HMI tags "2080SP242U01"
   "2080SP242U01.AI1" : Real AT %DB4304.DBD6, 500 ms
   "2080SP242U01.AI2" : Real AT %DB4304.DBD10, 500 ms
   "2080SP242U01.AI3" : Real AT %DB4304.DBD14, 500 ms
   "2080SP242U01.AO1a" : Real AT %DB4304.DBD34, 500 ms
   "2080SP242U01.AO1b" : Real AT %DB4304.DBD38, 500 ms
   "2080SP242U01.AO2a" : Real AT %DB4304.DBD42, 500 ms
   "2080SP242U01.AO2b" : Real AT %DB4304.DBD42, 500 ms
   "2080SP242U01.AO3a" : Real AT %DB4304.DBD50, 500 ms
   "2080SP242U01.AO3b" : Real AT %DB4304.DBD46, 500 ms
   "2080SP242U01.BlockInfo" : Array [0..4] of Int AT %DB4304.DBX74.0, 500 ms
   "2080SP242U01.DefaultText" : TextRef, internal   // Заголовок POPUP окна. При експорте из ECS через скрипт заполняется автоматически, если теги копируются в ручную то требуется в ручную задатать свойство Start Value
   "2080SP242U01.DI.ACK" : Bool AT %DB4304.DBX5.3, 500 ms
   "2080SP242U01.DI.ASTR" : Bool AT %DB4304.DBX2.1, 500 ms
   "2080SP242U01.DI.BUSF" : Bool AT %DB4304.DBX4.5, 500 ms
   "2080SP242U01.DI.DIR" : Bool AT %DB4304.DBX2.2, 500 ms
   "2080SP242U01.DI.DOPR" : Bool AT %DB4304.DBX4.6, 500 ms
   "2080SP242U01.DI.DRDY" : Bool AT %DB4304.DBX3.6, 500 ms
   "2080SP242U01.DI.DTEST" : Bool AT %DB4304.DBX4.7, 500 ms
   "2080SP242U01.DI.EARTH" : Bool AT %DB4304.DBX4.1, 500 ms
   "2080SP242U01.DI.ES" : Bool AT %DB4304.DBX5.2, 500 ms
   "2080SP242U01.DI.GFA" : Bool AT %DB4304.DBX4.3, 500 ms
   "2080SP242U01.DI.GWA" : Bool AT %DB4304.DBX4.4, 500 ms
   "2080SP242U01.DI.LSTP" : Bool AT %DB4304.DBX3.2, 500 ms
   "2080SP242U01.DI.LSTR1" : Bool AT %DB4304.DBX3.0, 500 ms
   "2080SP242U01.DI.LSTR2" : Bool AT %DB4304.DBX3.1, 500 ms
   "2080SP242U01.DI.MCC" : Bool AT %DB4304.DBX2.3, 500 ms
   "2080SP242U01.DI.MD" : Bool AT %DB4304.DBX3.7, 500 ms
   "2080SP242U01.DI.OVL" : Bool AT %DB4304.DBX2.5, 500 ms
   "2080SP242U01.DI.RDY" : Bool AT %DB4304.DBX2.4, 500 ms
   "2080SP242U01.DI.REM" : Bool AT %DB4304.DBX3.3, 500 ms
   "2080SP242U01.DI.RET1" : Bool AT %DB4304.DBX2.6, 500 ms
   "2080SP242U01.DI.RET2" : Bool AT %DB4304.DBX2.7, 500 ms
   "2080SP242U01.DI.SEL" : Bool AT %DB4304.DBX2.0, 500 ms
   "2080SP242U01.DI.SFS" : Bool AT %DB4304.DBX5.0, 500 ms
   "2080SP242U01.DI.SLS" : Bool AT %DB4304.DBX5.1, 500 ms
   "2080SP242U01.DI.SSW" : Bool AT %DB4304.DBX3.4, 500 ms
   "2080SP242U01.DI.STALL" : Bool AT %DB4304.DBX4.0, 500 ms
   "2080SP242U01.DI.TFA" : Bool AT %DB4304.DBX3.5, 500 ms
   "2080SP242U01.DI.UBAL" : Bool AT %DB4304.DBX4.2, 500 ms
   "2080SP242U01.DQ.ASTW" : Bool AT %DB4304.DBX32.0, 500 ms
   "2080SP242U01.DQ.AUT" : Bool AT %DB4304.DBX31.4, 500 ms
   "2080SP242U01.DQ.CON1" : Bool AT %DB4304.DBX30.0, 500 ms
   "2080SP242U01.DQ.CON2" : Bool AT %DB4304.DBX30.1, 500 ms
   "2080SP242U01.DQ.LAMP1" : Bool AT %DB4304.DBX30.2, 500 ms
   "2080SP242U01.DQ.LAMP2" : Bool AT %DB4304.DBX30.3, 500 ms
   "2080SP242U01.DQ.LOC" : Bool AT %DB4304.DBX31.2, 500 ms
   "2080SP242U01.DQ.MAN" : Bool AT %DB4304.DBX31.3, 500 ms
   "2080SP242U01.DQ.OK" : Bool AT %DB4304.DBX31.1, 500 ms
   "2080SP242U01.DQ.RD1" : Bool AT %DB4304.DBX30.5, 500 ms
   "2080SP242U01.DQ.RD2" : Bool AT %DB4304.DBX30.6, 500 ms
   "2080SP242U01.DQ.RES" : Bool AT %DB4304.DBX31.6, 500 ms
   "2080SP242U01.DQ.RUN1" : Bool AT %DB4304.DBX30.7, 500 ms
   "2080SP242U01.DQ.RUN2" : Bool AT %DB4304.DBX31.0, 500 ms
   "2080SP242U01.DQ.SACK" : Bool AT %DB4304.DBX30.4, 500 ms
   "2080SP242U01.DQ.SS" : Bool AT %DB4304.DBX31.5, 500 ms
   "2080SP242U01.DQ.TESTP" : Bool AT %DB4304.DBX31.7, 500 ms
   "2080SP242U01.FP_CMD" : Int AT %DB4304.DBW84, 500 ms
   "2080SP242U01.FP_CMD.AckAlarm" : Bool AT %DB4304.DBX84.7, 500 ms
   "2080SP242U01.FP_CMD.Auto" : Bool AT %DB4304.DBX85.0, 500 ms
   "2080SP242U01.FP_CMD.Local" : Bool AT %DB4304.DBX85.2, 500 ms
   "2080SP242U01.FP_CMD.Manual" : Bool AT %DB4304.DBX85.1, 500 ms
   "2080SP242U01.FP_CMD.QuickStop" : Bool AT %DB4304.DBX84.0, 500 ms
   "2080SP242U01.FP_CMD.Reset" : Bool AT %DB4304.DBX85.6, 500 ms
   "2080SP242U01.FP_CMD.Start1" : Bool AT %DB4304.DBX85.3, 500 ms
   "2080SP242U01.FP_CMD.Start2" : Bool AT %DB4304.DBX85.4, 500 ms
   "2080SP242U01.FP_CMD.Stop" : Bool AT %DB4304.DBX85.5, 500 ms
   "2080SP242U01.FP_CMD.Test" : Bool AT %DB4304.DBX85.7, 500 ms
   "2080SP242U01.FP_DIM.Auto" : Bool AT %DB4304.DBX92.0, 500 ms
   "2080SP242U01.FP_DIM.FP_DIM" : Bool AT %DB4304.DBX92.0, 500 ms
   "2080SP242U01.FP_DIM.Local" : Bool AT %DB4304.DBX92.1, 500 ms
   "2080SP242U01.FP_DIM.Manual" : Bool AT %DB4304.DBX92.2, 500 ms
   "2080SP242U01.FP_DIM.QStop" : Bool AT %DB4304.DBX92.7, 500 ms
   "2080SP242U01.FP_DIM.Reset" : Bool AT %DB4304.DBX93.0, 500 ms
   "2080SP242U01.FP_DIM.Start1" : Bool AT %DB4304.DBX92.3, 500 ms
   "2080SP242U01.FP_DIM.Start2" : Bool AT %DB4304.DBX92.4, 500 ms
   "2080SP242U01.FP_DIM.Stop" : Bool AT %DB4304.DBX92.5, 500 ms
   "2080SP242U01.FP_DIM.TEst" : Bool AT %DB4304.DBX92.6, 500 ms
   "2080SP242U01.FP_DIM1" : Array [0..15] of Bool AT %DB4304.DBX92.0, 500 ms
   "2080SP242U01.FP_EN.Mode_Auto" : Bool AT %DB4304.DBX90.0, 500 ms
   "2080SP242U01.FP_EN.Mode_Loc" : Bool AT %DB4304.DBX90.2, 500 ms
   "2080SP242U01.FP_EN.Mode_Loc_1" : Bool AT %DB4304.DBX90.3, 500 ms
   "2080SP242U01.FP_EN.Mode_Man" : Bool AT %DB4304.DBX90.1, 500 ms
   "2080SP242U01.FP_EN.Mode_SS_Field" : Bool AT %DB4304.DBX90.4, 500 ms
   "2080SP242U01.FP_EN.Mode_SS_FP" : Bool AT %DB4304.DBX90.5, 500 ms
   "2080SP242U01.FP_EN.Mode_Test" : Bool AT %DB4304.DBX90.3, 500 ms
   "2080SP242U01.FP_EN.PB_QStop" : Bool AT %DB4304.DBX90.6, 500 ms
   "2080SP242U01.FP_PARM.AI1_Max" : Real AT %DB4304.DBD158, 500 ms
   "2080SP242U01.FP_PARM.AI1_Min" : Real AT %DB4304.DBD162, 500 ms
   "2080SP242U01.FP_PARM.AI2_Max" : Real AT %DB4304.DBD166, 500 ms
   "2080SP242U01.FP_PARM.AI2_Min" : Real AT %DB4304.DBD170, 500 ms
   "2080SP242U01.FP_PARM.AI3_Max" : Real AT %DB4304.DBD174, 500 ms
   "2080SP242U01.FP_PARM.AI3_Min" : Real AT %DB4304.DBD178, 500 ms
   "2080SP242U01.FP_PARM.AO1a_Max" : Real AT %DB4304.DBD182, 500 ms
   "2080SP242U01.FP_PARM.AO1a_Min" : Real AT %DB4304.DBD186, 500 ms
   "2080SP242U01.FP_PARM.AO1b_Max" : Real AT %DB4304.DBD206, 500 ms
   "2080SP242U01.FP_PARM.AO1b_Min" : Real AT %DB4304.DBD210, 500 ms
   "2080SP242U01.FP_PARM.AO2a_Max" : Real AT %DB4304.DBD190, 500 ms
   "2080SP242U01.FP_PARM.AO2a_Min" : Real AT %DB4304.DBD194, 500 ms
   "2080SP242U01.FP_PARM.AO2b_Max" : Real AT %DB4304.DBD214, 500 ms
   "2080SP242U01.FP_PARM.AO2b_Min" : Real AT %DB4304.DBD218, 500 ms
   "2080SP242U01.FP_PARM.AO3a_Max" : Real AT %DB4304.DBD198, 500 ms
   "2080SP242U01.FP_PARM.AO3a_Min" : Real AT %DB4304.DBD202, 500 ms
   "2080SP242U01.FP_PARM.AO3b_Max" : Real AT %DB4304.DBD222, 500 ms
   "2080SP242U01.FP_PARM.AO3b_Min" : Real AT %DB4304.DBD226, 500 ms
   "2080SP242U01.FP_PARM.ChangeDir_Acc" : Int AT %DB4304.DBW138, 500 ms
   "2080SP242U01.FP_PARM.ChangeDir_Pre" : Int AT %DB4304.DBW136, 500 ms
   "2080SP242U01.FP_PARM.DelayStart_Acc" : Int AT %DB4304.DBW114, 500 ms
   "2080SP242U01.FP_PARM.DelayStart_Pre" : Int AT %DB4304.DBW112, 500 ms
   "2080SP242U01.FP_PARM.DelayStop_Acc" : Int AT %DB4304.DBW118, 500 ms
   "2080SP242U01.FP_PARM.DelayStop_Pre" : Int AT %DB4304.DBW116, 500 ms
   "2080SP242U01.FP_PARM.INTL" : Bool AT %DB4304.DBX230.0, 500 ms
   "2080SP242U01.FP_PARM.INTL_SEQ_STP" : Bool AT %DB4304.DBX230.3, 500 ms
   "2080SP242U01.FP_PARM.INTL_SEQ_STR1" : Bool AT %DB4304.DBX230.1, 500 ms
   "2080SP242U01.FP_PARM.INTL_SEQ_STR2" : Bool AT %DB4304.DBX230.2, 500 ms
   "2080SP242U01.FP_PARM.LeaveFS_Acc" : Int AT %DB4304.DBW142, 500 ms
   "2080SP242U01.FP_PARM.LeaveFS_Pre" : Int AT %DB4304.DBW140, 500 ms
   "2080SP242U01.FP_PARM.MD_Freq_PV" : Int AT %DB4304.DBW154, 500 ms
   "2080SP242U01.FP_PARM.MD_Freq_SP" : Int AT %DB4304.DBW152, 500 ms
   "2080SP242U01.FP_PARM.ReachFS_Acc" : Int AT %DB4304.DBW150, 500 ms
   "2080SP242U01.FP_PARM.ReachFS_Pre" : Int AT %DB4304.DBW148, 500 ms
   "2080SP242U01.FP_PARM.ReachLS_Acc" : Int AT %DB4304.DBW146, 500 ms
   "2080SP242U01.FP_PARM.ReachLS_Pre" : Int AT %DB4304.DBW144, 500 ms
   "2080SP242U01.FP_PARM.ReturnMon_Acc" : Int AT %DB4304.DBW122, 500 ms
   "2080SP242U01.FP_PARM.ReturnMon_Pre" : Int AT %DB4304.DBW120, 500 ms
   "2080SP242U01.FP_PARM.RunDelay1_Acc" : Int AT %DB4304.DBW106, 500 ms
   "2080SP242U01.FP_PARM.RunDelay1_Pre" : Int AT %DB4304.DBW104, 500 ms
   "2080SP242U01.FP_PARM.RunDelay2_Acc" : Int AT %DB4304.DBW110, 500 ms
   "2080SP242U01.FP_PARM.RunDelay2_Pre" : Int AT %DB4304.DBW108, 500 ms
   "2080SP242U01.FP_PARM.SpeedMonOffDelay_Acc" : Int AT %DB4304.DBW130, 500 ms
   "2080SP242U01.FP_PARM.SpeedMonOffDelay_Pre" : Int AT %DB4304.DBW128, 500 ms
   "2080SP242U01.FP_PARM.SpeedMonOnDelay_Acc" : Int AT %DB4304.DBW126, 500 ms
   "2080SP242U01.FP_PARM.SpeedMonOnDelay_Pre" : Int AT %DB4304.DBW124, 500 ms
   "2080SP242U01.FP_PARM.SpeedMonTrigDelay_Acc" : Int AT %DB4304.DBW134, 500 ms
   "2080SP242U01.FP_PARM.SpeedMonTrigDelay_Pre" : Int AT %DB4304.DBW132, 500 ms
   "2080SP242U01.FP_PARM.StartWarn_Acc" : Int AT %DB4304.DBW102, 500 ms
   "2080SP242U01.FP_PARM.StartWarn_Pre" : Int AT %DB4304.DBW100, 500 ms
   "2080SP242U01.FP_PARM.StopReason" : Int AT %DB4304.DBW156, 500 ms
   "2080SP242U01.FP_SEL.INCH_Loc" : Bool AT %DB4304.DBX87.7, 500 ms
   "2080SP242U01.FP_SEL.INCH_Man" : Bool AT %DB4304.DBX87.6, 500 ms
   "2080SP242U01.FP_SEL.MD" : Bool AT %DB4304.DBX86.0, 500 ms
   "2080SP242U01.FP_SEL.MD_Maintain" : Bool AT %DB4304.DBX86.3, 500 ms
   "2080SP242U01.FP_SEL.MD_OnOff" : Bool AT %DB4304.DBX86.2, 500 ms
   "2080SP242U01.FP_SEL.MD_Puls" : Bool AT %DB4304.DBX86.1, 500 ms
   "2080SP242U01.FP_SEL.MotorStarter" : Bool AT %DB4304.DBX87.3, 500 ms
   "2080SP242U01.FP_SEL.OutOfSevice" : Bool AT %DB4304.DBX88.0, 500 ms
   "2080SP242U01.FP_SEL.ParentCollection" : Bool AT %DB4304.DBX87.5, 500 ms
   "2080SP242U01.FP_SEL.ParentSupress" : Bool AT %DB4304.DBX87.4, 500 ms
   "2080SP242U01.FP_SEL.STW_AutoStart" : Bool AT %DB4304.DBX86.4, 500 ms
   "2080SP242U01.FP_SEL.STW_Local" : Bool AT %DB4304.DBX86.5, 500 ms
   "2080SP242U01.FP_SEL.STW_Manual" : Bool AT %DB4304.DBX86.6, 500 ms
   "2080SP242U01.FP_SEL.STW_Single" : Bool AT %DB4304.DBX86.7, 500 ms
   "2080SP242U01.FP_SEL.Type_Bimotor" : Bool AT %DB4304.DBX87.1, 500 ms
   "2080SP242U01.FP_SEL.Type_Indication" : Bool AT %DB4304.DBX87.2, 500 ms
   "2080SP242U01.FP_SEL.Type_Unimotor" : Bool AT %DB4304.DBX87.0, 500 ms
   "2080SP242U01.FP_SEL.WarningDrive" : Bool AT %DB4304.DBX88.1, 500 ms
   "2080SP242U01.FP_SHOW.ACK" : Bool AT %DB4304.DBX97.5, 500 ms
   "2080SP242U01.FP_SHOW.AI1" : Bool AT %DB4304.DBX95.0, 500 ms
   "2080SP242U01.FP_SHOW.AI2" : Bool AT %DB4304.DBX95.1, 500 ms
   "2080SP242U01.FP_SHOW.AI3" : Bool AT %DB4304.DBX95.2, 500 ms
   "2080SP242U01.FP_SHOW.ASTR" : Bool AT %DB4304.DBX99.2, 500 ms
   "2080SP242U01.FP_SHOW.B1" : Byte AT %DB4304.DBB95, 500 ms
   "2080SP242U01.FP_SHOW.B2" : Byte AT %DB4304.DBB96, 500 ms
   "2080SP242U01.FP_SHOW.B3" : Byte AT %DB4304.DBB97, 500 ms
   "2080SP242U01.FP_SHOW.B4" : Byte AT %DB4304.DBB98, 500 ms
   "2080SP242U01.FP_SHOW.BUSF" : Bool AT %DB4304.DBX97.2, 500 ms
   "2080SP242U01.FP_SHOW.ChangeDir" : Bool AT %DB4304.DBX99.0, 500 ms
   "2080SP242U01.FP_SHOW.CON2" : Bool AT %DB4304.DBX98.2, 500 ms
   "2080SP242U01.FP_SHOW.DelayRun2" : Bool AT %DB4304.DBX98.7, 500 ms
   "2080SP242U01.FP_SHOW.DOPR" : Bool AT %DB4304.DBX97.3, 500 ms
   "2080SP242U01.FP_SHOW.DRDY" : Bool AT %DB4304.DBX96.4, 500 ms
   "2080SP242U01.FP_SHOW.DTEST" : Bool AT %DB4304.DBX97.4, 500 ms
   "2080SP242U01.FP_SHOW.EARTH" : Bool AT %DB4304.DBX96.6, 500 ms
   "2080SP242U01.FP_SHOW.ES" : Bool AT %DB4304.DBX96.2, 500 ms
   "2080SP242U01.FP_SHOW.GFA" : Bool AT %DB4304.DBX97.0, 500 ms
   "2080SP242U01.FP_SHOW.GWA" : Bool AT %DB4304.DBX97.1, 500 ms
   "2080SP242U01.FP_SHOW.LSTP" : Bool AT %DB4304.DBX95.7, 500 ms
   "2080SP242U01.FP_SHOW.LSTR1" : Bool AT %DB4304.DBX97.6, 500 ms
   "2080SP242U01.FP_SHOW.LSTR2" : Bool AT %DB4304.DBX97.7, 500 ms
   "2080SP242U01.FP_SHOW.MCC" : Bool AT %DB4304.DBX95.4, 500 ms
   "2080SP242U01.FP_SHOW.MD" : Bool AT %DB4304.DBX98.6, 500 ms
   "2080SP242U01.FP_SHOW.OVL" : Bool AT %DB4304.DBX95.6, 500 ms
   "2080SP242U01.FP_SHOW.PB_Auto" : Bool AT %DB4304.DBX94.0, 500 ms
   "2080SP242U01.FP_SHOW.PB_Local" : Bool AT %DB4304.DBX94.1, 500 ms
   "2080SP242U01.FP_SHOW.PB_Manual" : Bool AT %DB4304.DBX94.2, 500 ms
   "2080SP242U01.FP_SHOW.PB_QStop" : Bool AT %DB4304.DBX94.7, 500 ms
   "2080SP242U01.FP_SHOW.PB_Reset" : Bool AT %DB4304.DBX99.1, 500 ms
   "2080SP242U01.FP_SHOW.PB_Start1" : Bool AT %DB4304.DBX94.3, 500 ms
   "2080SP242U01.FP_SHOW.PB_Start2" : Bool AT %DB4304.DBX94.4, 500 ms
   "2080SP242U01.FP_SHOW.PB_Stop" : Bool AT %DB4304.DBX94.5, 500 ms
   "2080SP242U01.FP_SHOW.PB_Test" : Bool AT %DB4304.DBX94.6, 500 ms
   "2080SP242U01.FP_SHOW.RD2" : Bool AT %DB4304.DBX98.3, 500 ms
   "2080SP242U01.FP_SHOW.RDY" : Bool AT %DB4304.DBX95.5, 500 ms
   "2080SP242U01.FP_SHOW.REM" : Bool AT %DB4304.DBX96.0, 500 ms
   "2080SP242U01.FP_SHOW.RET2" : Bool AT %DB4304.DBX98.0, 500 ms
   "2080SP242U01.FP_SHOW.RUN2" : Bool AT %DB4304.DBX98.1, 500 ms
   "2080SP242U01.FP_SHOW.SFS" : Bool AT %DB4304.DBX98.4, 500 ms
   "2080SP242U01.FP_SHOW.SLS" : Bool AT %DB4304.DBX98.5, 500 ms
   "2080SP242U01.FP_SHOW.SP" : Bool AT %DB4304.DBX95.3, 500 ms
   "2080SP242U01.FP_SHOW.SSW" : Bool AT %DB4304.DBX96.1, 500 ms
   "2080SP242U01.FP_SHOW.STALL" : Bool AT %DB4304.DBX96.5, 500 ms
   "2080SP242U01.FP_SHOW.TFA" : Bool AT %DB4304.DBX96.3, 500 ms
   "2080SP242U01.FP_SHOW.UBAL" : Bool AT %DB4304.DBX96.7, 500 ms
   "2080SP242U01.ModePointer" : Int AT %DB4304.DBW496, 500 ms
   "2080SP242U01.MSW" : DWord AT %DB4304.DBD62, 500 ms
   "2080SP242U01.ParentInfo" : TextRef, internal   // Имя родителя для попап окна, вкладка инфо. При експорте из ECS через скрипт заполняется автоматически, если теги копируются в ручную то требуется в ручную задатать свойство Start Value
   "2080SP242U01.SPSET" : Real AT %DB4304.DBD18, 500 ms
   "2080SP242U01.StatusWork" : Int AT %DB4304.DBW494, 500 ms

HMI tags "2900RS001A01F01"
   "2900RS001A01F01.MSW" : 52809b66-421d-457f-8884-6f7a49d4e247 AT %DB5013.DBX18.0, 500 ms
   "2900RS001A01F01.DefaultText" : TextRef, internal   // Заголовок POPUP окна. При експорте из ECS через скрипт заполняется автоматически, если теги копируются в ручную то требуется в ручную задатать свойство Start Value
   "2900RS001A01F01.BlockInfo" : Array [0..2] of Int AT %DB5013.DBX38.0, 500 ms
   "2900RS001A01F01.StatusWork" : Int AT %DB5013.DBW242, 500 ms
   "2900RS001A01F01.FP_PARAM.DampingTime" : Int AT %DB5013.DBW50, 500 ms
   "2900RS001A01F01.FP_PARAM.Force_Value" : Real AT %DB5013.DBD52, 500 ms
   "2900RS001A01F01.FP_PARAM.Scale_Min" : Real AT %DB5013.DBD56, 500 ms
   "2900RS001A01F01.FP_PARAM.Scale_Max" : Real AT %DB5013.DBD60, 500 ms
   "2900RS001A01F01.FP_PARAM.Gradient" : Real AT %DB5013.DBD64, 500 ms
   "2900RS001A01F01.FP_PARAM.Grad_Pos" : Real AT %DB5013.DBD68, 500 ms
   "2900RS001A01F01.FP_PARAM.Grad_Neg" : Real AT %DB5013.DBD72, 500 ms
   "2900RS001A01F01.FP_PARAM.Grad_X" : Real AT %DB5013.DBD76, 500 ms
   "2900RS001A01F01.FP_PARAM.Gradient_Time_Pre" : Int AT %DB5013.DBW80, 500 ms
   "2900RS001A01F01.FP_PARAM.Gradient_Time_ACC" : Int AT %DB5013.DBW82, 500 ms
   "2900RS001A01F01.FP_PARAM.Alarm_Hyst" : Real AT %DB5013.DBD84, 500 ms
   "2900RS001A01F01.FP_PARAM.AlarmLimit_H3" : Real AT %DB5013.DBD88, 500 ms
   "2900RS001A01F01.FP_PARAM.AlarmLimit_H2" : Real AT %DB5013.DBD92, 500 ms
   "2900RS001A01F01.FP_PARAM.AlarmLimit_H1" : Real AT %DB5013.DBD96, 500 ms
   "2900RS001A01F01.FP_PARAM.AlarmLimit_L1" : Real AT %DB5013.DBD100, 500 ms
   "2900RS001A01F01.FP_PARAM.AlarmLimit_L2" : Real AT %DB5013.DBD104, 500 ms
   "2900RS001A01F01.FP_PARAM.AlarmLimit_L3" : Real AT %DB5013.DBD108, 500 ms
   "2900RS001A01F01.FP_PARAM.AlarmDelay_H3_Pre" : Int AT %DB5013.DBW112, 500 ms
   "2900RS001A01F01.FP_PARAM.AlarmDelay_H3_Acc" : Int AT %DB5013.DBW114, 500 ms
   "2900RS001A01F01.FP_PARAM.AlarmDelay_H2_Pre" : Int AT %DB5013.DBW116, 500 ms
   "2900RS001A01F01.FP_PARAM.AlarmDelay_H2_Acc" : Int AT %DB5013.DBW118, 500 ms
   "2900RS001A01F01.FP_PARAM.AlarmDelay_H1_Pre" : Int AT %DB5013.DBW120, 500 ms
   "2900RS001A01F01.FP_PARAM.AlarmDelay_H1_Acc" : Int AT %DB5013.DBW122, 500 ms
   "2900RS001A01F01.FP_PARAM.AlarmDelay_L1_Pre" : Int AT %DB5013.DBW124, 500 ms
   "2900RS001A01F01.FP_PARAM.AlarmDelay_L1_Acc" : Int AT %DB5013.DBW126, 500 ms
   "2900RS001A01F01.FP_PARAM.AlarmDelay_L2_Pre" : Int AT %DB5013.DBW128, 500 ms
   "2900RS001A01F01.FP_PARAM.AlarmDelay_L2_Acc" : Int AT %DB5013.DBW130, 500 ms
   "2900RS001A01F01.FP_PARAM.AlarmDelay_L3_Pre" : Int AT %DB5013.DBW132, 500 ms
   "2900RS001A01F01.FP_PARAM.AlarmDelay_L3_Acc" : Int AT %DB5013.DBW134, 500 ms
   "2900RS001A01F01.FP_PARAM.OpenLoopDelay_Pre" : Int AT %DB5013.DBW136, 500 ms
   "2900RS001A01F01.FP_PARAM.OpenLoopDelay_Acc" : Int AT %DB5013.DBW138, 500 ms
   "2900RS001A01F01.FP_PARAM.OverRangeDelay_Pre" : Int AT %DB5013.DBW140, 500 ms
   "2900RS001A01F01.FP_PARAM.OverRangeDelay_Acc" : Int AT %DB5013.DBW142, 500 ms
   "2900RS001A01F01.FP_PARAM.AuxLimit_H2_Value" : Real AT %DB5013.DBD144, 500 ms
   "2900RS001A01F01.FP_PARAM.AuxLimit_H1_Value" : Real AT %DB5013.DBD148, 500 ms
   "2900RS001A01F01.FP_PARAM.AuxLimit_L2_Value" : Real AT %DB5013.DBD152, 500 ms
   "2900RS001A01F01.FP_PARAM.AuxLimit_L1_Value" : Real AT %DB5013.DBD156, 500 ms
   "2900RS001A01F01.Unit" : TextRef, internal   // Еденицы измерения При експорте из ECS через скрипт заполняется автоматически, если теги копируются в ручную то требуется задатать свойство Text
   "2900RS001A01F01.Decimals" : TextRef, internal   // Формат отображения При експорте из ECS через скрипт, заполняется автоматически. Если теги копируются в ручную то требуется задатать свойство Text s999999.9
   "2900RS001A01F01.FP_EN.Square" : Bool AT %DB5013.DBX46.0, 500 ms
   "2900RS001A01F01.FP_EN.SquareRoot" : Bool AT %DB5013.DBX46.1, 500 ms
   "2900RS001A01F01.FP_EN.ParentSupress" : Bool AT %DB5013.DBX46.2, 500 ms
   "2900RS001A01F01.FP_EN.ParentSupressUnit" : Bool AT %DB5013.DBX46.3, 500 ms
   "2900RS001A01F01.FP_EN.Force" : Bool AT %DB5013.DBX46.4, 500 ms
   "2900RS001A01F01.FP_EN.Damping" : Bool AT %DB5013.DBX46.5, 500 ms
   "2900RS001A01F01.FP_EN.Gradient_Pos" : Bool AT %DB5013.DBX46.6, 500 ms
   "2900RS001A01F01.FP_EN.Gradient_Neg" : Bool AT %DB5013.DBX46.7, 500 ms
   "2900RS001A01F01.FP_EN.Hysteresis" : Bool AT %DB5013.DBX47.0, 500 ms
   "2900RS001A01F01.FP_EN.Alarm_H3" : Bool AT %DB5013.DBX47.1, 500 ms
   "2900RS001A01F01.FP_EN.Alarm_H2" : Bool AT %DB5013.DBX47.2, 500 ms
   "2900RS001A01F01.FP_EN.Alarm_H1" : Bool AT %DB5013.DBX47.3, 500 ms
   "2900RS001A01F01.FP_EN.Alarm_L1" : Bool AT %DB5013.DBX47.4, 500 ms
   "2900RS001A01F01.FP_EN.Alarm_L2" : Bool AT %DB5013.DBX47.5, 500 ms
   "2900RS001A01F01.FP_EN.Alarm_L3" : Bool AT %DB5013.DBX47.6, 500 ms
   "2900RS001A01F01.FP_EN.AlarmDelay_H3" : Bool AT %DB5013.DBX47.7, 500 ms
   "2900RS001A01F01.FP_EN.AlarmDelay_H2" : Bool AT %DB5013.DBX48.0, 500 ms
   "2900RS001A01F01.FP_EN.AlarmDelay_H1" : Bool AT %DB5013.DBX48.1, 500 ms
   "2900RS001A01F01.FP_EN.AlarmDelay_L1" : Bool AT %DB5013.DBX48.2, 500 ms
   "2900RS001A01F01.FP_EN.AlarmDelay_L2" : Bool AT %DB5013.DBX48.3, 500 ms
   "2900RS001A01F01.FP_EN.AlarmDelay_L3" : Bool AT %DB5013.DBX48.4, 500 ms
   "2900RS001A01F01.FP_EN.ROC_Warn" : Bool AT %DB5013.DBX48.5, 500 ms
   "2900RS001A01F01.FP_EN.U_Range_Warn" : Bool AT %DB5013.DBX48.6, 500 ms
   "2900RS001A01F01.FP_EN.O_Range_Warn" : Bool AT %DB5013.DBX48.7, 500 ms
   "2900RS001A01F01.trend_tag_name" : TextRef, internal   // Еденицы измерения При експорте из ECS через скрипт - заполняется автоматически, если теги копируются в ручную то требуется задатать свойство Text - имя тега для тренда
   "2900RS001A01F01.DQ.AL_H3" : Bool AT %DB5013.DBX16.0, 500 ms
   "2900RS001A01F01.DQ.AL_H2" : Bool AT %DB5013.DBX16.1, 500 ms
   "2900RS001A01F01.DQ.AL_H1" : Bool AT %DB5013.DBX16.2, 500 ms
   "2900RS001A01F01.DQ.AL_L1" : Bool AT %DB5013.DBX16.3, 500 ms
   "2900RS001A01F01.DQ.AL_L2" : Bool AT %DB5013.DBX16.4, 500 ms
   "2900RS001A01F01.DQ.AL_L3" : Bool AT %DB5013.DBX16.5, 500 ms
   "2900RS001A01F01.DQ.SIG_OK" : Bool AT %DB5013.DBX16.6, 500 ms
   "2900RS001A01F01.DQ.LIM_H2" : Bool AT %DB5013.DBX16.7, 500 ms
   "2900RS001A01F01.DQ.LIM_H1" : Bool AT %DB5013.DBX17.0, 500 ms
   "2900RS001A01F01.DQ.LIM_L1" : Bool AT %DB5013.DBX17.1, 500 ms
   "2900RS001A01F01.DQ.LIM_L2" : Bool AT %DB5013.DBX17.2, 500 ms
   "2900RS001A01F01.DQ.GR_P" : Bool AT %DB5013.DBX17.3, 500 ms
   "2900RS001A01F01.DQ.GR_N" : Bool AT %DB5013.DBX17.4, 500 ms
   "2900RS001A01F01.I.IN" : Real AT %DB5013.DBD2, 500 ms
   "2900RS001A01F01.I.SIG_TYPE" : Int AT %DB5013.DBW0, 500 ms
   "2900RS001A01F01.I.FI_BUS" : Byte AT %DB5013.DBB6, 500 ms
   "2900RS001A01F01.DI.U_RANGE" : Bool AT %DB5013.DBX7.0, 500 ms
   "2900RS001A01F01.DI.O_RANGE" : Bool AT %DB5013.DBX7.1, 500 ms
   "2900RS001A01F01.DI.SIG_FAULT" : Bool AT %DB5013.DBX7.2, 500 ms
   "2900RS001A01F01.DI.EnConfig" : Bool AT %DB5013.DBX7.3, 500 ms
   "2900RS001A01F01.DI.AEN" : Bool AT %DB5013.DBX7.4, 500 ms
   "2900RS001A01F01.DI.AL_SUPR" : Bool AT %DB5013.DBX7.5, 500 ms
   "2900RS001A01F01.Q.PV_NORM" : Real AT %DB5013.DBD8, 500 ms
   "2900RS001A01F01.Q.PV_SCAL" : Real AT %DB5013.DBD12, 500 ms
   "2900RS001A01F01.ParentInfo" : TextRef, internal   // Имя родителя для попап окна, вкладка инфо. При експорте из ECS через скрипт заполняется автоматически, если теги копируются в ручную то требуется в ручную задатать свойство Start Value

HMI tags "2900RS001A01F02"
   "2900RS001A01F02.MSW" : 52809b66-421d-457f-8884-6f7a49d4e247 AT %DB5014.DBX18.0, 500 ms
   "2900RS001A01F02.DefaultText" : TextRef, internal   // Заголовок POPUP окна. При експорте из ECS через скрипт заполняется автоматически, если теги копируются в ручную то требуется в ручную задатать свойство Start Value
   "2900RS001A01F02.BlockInfo" : Array [0..2] of Int AT %DB5014.DBX38.0, 500 ms
   "2900RS001A01F02.StatusWork" : Int AT %DB5014.DBW242, 500 ms
   "2900RS001A01F02.FP_PARAM.DampingTime" : Int AT %DB5014.DBW50, 500 ms
   "2900RS001A01F02.FP_PARAM.Force_Value" : Real AT %DB5014.DBD52, 500 ms
   "2900RS001A01F02.FP_PARAM.Scale_Min" : Real AT %DB5014.DBD56, 500 ms
   "2900RS001A01F02.FP_PARAM.Scale_Max" : Real AT %DB5014.DBD60, 500 ms
   "2900RS001A01F02.FP_PARAM.Gradient" : Real AT %DB5014.DBD64, 500 ms
   "2900RS001A01F02.FP_PARAM.Grad_Pos" : Real AT %DB5014.DBD68, 500 ms
   "2900RS001A01F02.FP_PARAM.Grad_Neg" : Real AT %DB5014.DBD72, 500 ms
   "2900RS001A01F02.FP_PARAM.Grad_X" : Real AT %DB5014.DBD76, 500 ms
   "2900RS001A01F02.FP_PARAM.Gradient_Time_Pre" : Int AT %DB5014.DBW80, 500 ms
   "2900RS001A01F02.FP_PARAM.Gradient_Time_ACC" : Int AT %DB5014.DBW82, 500 ms
   "2900RS001A01F02.FP_PARAM.Alarm_Hyst" : Real AT %DB5014.DBD84, 500 ms
   "2900RS001A01F02.FP_PARAM.AlarmLimit_H3" : Real AT %DB5014.DBD88, 500 ms
   "2900RS001A01F02.FP_PARAM.AlarmLimit_H2" : Real AT %DB5014.DBD92, 500 ms
   "2900RS001A01F02.FP_PARAM.AlarmLimit_H1" : Real AT %DB5014.DBD96, 500 ms
   "2900RS001A01F02.FP_PARAM.AlarmLimit_L1" : Real AT %DB5014.DBD100, 500 ms
   "2900RS001A01F02.FP_PARAM.AlarmLimit_L2" : Real AT %DB5014.DBD104, 500 ms
   "2900RS001A01F02.FP_PARAM.AlarmLimit_L3" : Real AT %DB5014.DBD108, 500 ms
   "2900RS001A01F02.FP_PARAM.AlarmDelay_H3_Pre" : Int AT %DB5014.DBW112, 500 ms
   "2900RS001A01F02.FP_PARAM.AlarmDelay_H3_Acc" : Int AT %DB5014.DBW114, 500 ms
   "2900RS001A01F02.FP_PARAM.AlarmDelay_H2_Pre" : Int AT %DB5014.DBW116, 500 ms
   "2900RS001A01F02.FP_PARAM.AlarmDelay_H2_Acc" : Int AT %DB5014.DBW118, 500 ms
   "2900RS001A01F02.FP_PARAM.AlarmDelay_H1_Pre" : Int AT %DB5014.DBW120, 500 ms
   "2900RS001A01F02.FP_PARAM.AlarmDelay_H1_Acc" : Int AT %DB5014.DBW122, 500 ms
   "2900RS001A01F02.FP_PARAM.AlarmDelay_L1_Pre" : Int AT %DB5014.DBW124, 500 ms
   "2900RS001A01F02.FP_PARAM.AlarmDelay_L1_Acc" : Int AT %DB5014.DBW126, 500 ms
   "2900RS001A01F02.FP_PARAM.AlarmDelay_L2_Pre" : Int AT %DB5014.DBW128, 500 ms
   "2900RS001A01F02.FP_PARAM.AlarmDelay_L2_Acc" : Int AT %DB5014.DBW130, 500 ms
   "2900RS001A01F02.FP_PARAM.AlarmDelay_L3_Pre" : Int AT %DB5014.DBW132, 500 ms
   "2900RS001A01F02.FP_PARAM.AlarmDelay_L3_Acc" : Int AT %DB5014.DBW134, 500 ms
   "2900RS001A01F02.FP_PARAM.OpenLoopDelay_Pre" : Int AT %DB5014.DBW136, 500 ms
   "2900RS001A01F02.FP_PARAM.OpenLoopDelay_Acc" : Int AT %DB5014.DBW138, 500 ms
   "2900RS001A01F02.FP_PARAM.OverRangeDelay_Pre" : Int AT %DB5014.DBW140, 500 ms
   "2900RS001A01F02.FP_PARAM.OverRangeDelay_Acc" : Int AT %DB5014.DBW142, 500 ms
   "2900RS001A01F02.FP_PARAM.AuxLimit_H2_Value" : Real AT %DB5014.DBD144, 500 ms
   "2900RS001A01F02.FP_PARAM.AuxLimit_H1_Value" : Real AT %DB5014.DBD148, 500 ms
   "2900RS001A01F02.FP_PARAM.AuxLimit_L2_Value" : Real AT %DB5014.DBD152, 500 ms
   "2900RS001A01F02.FP_PARAM.AuxLimit_L1_Value" : Real AT %DB5014.DBD156, 500 ms
   "2900RS001A01F02.Unit" : TextRef, internal   // Еденицы измерения При експорте из ECS через скрипт заполняется автоматически, если теги копируются в ручную то требуется задатать свойство Text
   "2900RS001A01F02.Decimals" : TextRef, internal   // Формат отображения При експорте из ECS через скрипт, заполняется автоматически. Если теги копируются в ручную то требуется задатать свойство Text s999999.9
   "2900RS001A01F02.FP_EN.Square" : Bool AT %DB5014.DBX46.0, 500 ms
   "2900RS001A01F02.FP_EN.SquareRoot" : Bool AT %DB5014.DBX46.1, 500 ms
   "2900RS001A01F02.FP_EN.ParentSupress" : Bool AT %DB5014.DBX46.2, 500 ms
   "2900RS001A01F02.FP_EN.ParentSupressUnit" : Bool AT %DB5014.DBX46.3, 500 ms
   "2900RS001A01F02.FP_EN.Force" : Bool AT %DB5014.DBX46.4, 500 ms
   "2900RS001A01F02.FP_EN.Damping" : Bool AT %DB5014.DBX46.5, 500 ms
   "2900RS001A01F02.FP_EN.Gradient_Pos" : Bool AT %DB5014.DBX46.6, 500 ms
   "2900RS001A01F02.FP_EN.Gradient_Neg" : Bool AT %DB5014.DBX46.7, 500 ms
   "2900RS001A01F02.FP_EN.Hysteresis" : Bool AT %DB5014.DBX47.0, 500 ms
   "2900RS001A01F02.FP_EN.Alarm_H3" : Bool AT %DB5014.DBX47.1, 500 ms
   "2900RS001A01F02.FP_EN.Alarm_H2" : Bool AT %DB5014.DBX47.2, 500 ms
   "2900RS001A01F02.FP_EN.Alarm_H1" : Bool AT %DB5014.DBX47.3, 500 ms
   "2900RS001A01F02.FP_EN.Alarm_L1" : Bool AT %DB5014.DBX47.4, 500 ms
   "2900RS001A01F02.FP_EN.Alarm_L2" : Bool AT %DB5014.DBX47.5, 500 ms
   "2900RS001A01F02.FP_EN.Alarm_L3" : Bool AT %DB5014.DBX47.6, 500 ms
   "2900RS001A01F02.FP_EN.AlarmDelay_H3" : Bool AT %DB5014.DBX47.7, 500 ms
   "2900RS001A01F02.FP_EN.AlarmDelay_H2" : Bool AT %DB5014.DBX48.0, 500 ms
   "2900RS001A01F02.FP_EN.AlarmDelay_H1" : Bool AT %DB5014.DBX48.1, 500 ms
   "2900RS001A01F02.FP_EN.AlarmDelay_L1" : Bool AT %DB5014.DBX48.2, 500 ms
   "2900RS001A01F02.FP_EN.AlarmDelay_L2" : Bool AT %DB5014.DBX48.3, 500 ms
   "2900RS001A01F02.FP_EN.AlarmDelay_L3" : Bool AT %DB5014.DBX48.4, 500 ms
   "2900RS001A01F02.FP_EN.ROC_Warn" : Bool AT %DB5014.DBX48.5, 500 ms
   "2900RS001A01F02.FP_EN.U_Range_Warn" : Bool AT %DB5014.DBX48.6, 500 ms
   "2900RS001A01F02.FP_EN.O_Range_Warn" : Bool AT %DB5014.DBX48.7, 500 ms
   "2900RS001A01F02.trend_tag_name" : TextRef, internal   // Еденицы измерения При експорте из ECS через скрипт - заполняется автоматически, если теги копируются в ручную то требуется задатать свойство Text - имя тега для тренда
   "2900RS001A01F02.DQ.AL_H3" : Bool AT %DB5014.DBX16.0, 500 ms
   "2900RS001A01F02.DQ.AL_H2" : Bool AT %DB5014.DBX16.1, 500 ms
   "2900RS001A01F02.DQ.AL_H1" : Bool AT %DB5014.DBX16.2, 500 ms
   "2900RS001A01F02.DQ.AL_L1" : Bool AT %DB5014.DBX16.3, 500 ms
   "2900RS001A01F02.DQ.AL_L2" : Bool AT %DB5014.DBX16.4, 500 ms
   "2900RS001A01F02.DQ.AL_L3" : Bool AT %DB5014.DBX16.5, 500 ms
   "2900RS001A01F02.DQ.SIG_OK" : Bool AT %DB5014.DBX16.6, 500 ms
   "2900RS001A01F02.DQ.LIM_H2" : Bool AT %DB5014.DBX16.7, 500 ms
   "2900RS001A01F02.DQ.LIM_H1" : Bool AT %DB5014.DBX17.0, 500 ms
   "2900RS001A01F02.DQ.LIM_L1" : Bool AT %DB5014.DBX17.1, 500 ms
   "2900RS001A01F02.DQ.LIM_L2" : Bool AT %DB5014.DBX17.2, 500 ms
   "2900RS001A01F02.DQ.GR_P" : Bool AT %DB5014.DBX17.3, 500 ms
   "2900RS001A01F02.DQ.GR_N" : Bool AT %DB5014.DBX17.4, 500 ms
   "2900RS001A01F02.I.IN" : Real AT %DB5014.DBD2, 500 ms
   "2900RS001A01F02.I.SIG_TYPE" : Int AT %DB5014.DBW0, 500 ms
   "2900RS001A01F02.I.FI_BUS" : Byte AT %DB5014.DBB6, 500 ms
   "2900RS001A01F02.DI.U_RANGE" : Bool AT %DB5014.DBX7.0, 500 ms
   "2900RS001A01F02.DI.O_RANGE" : Bool AT %DB5014.DBX7.1, 500 ms
   "2900RS001A01F02.DI.SIG_FAULT" : Bool AT %DB5014.DBX7.2, 500 ms
   "2900RS001A01F02.DI.EnConfig" : Bool AT %DB5014.DBX7.3, 500 ms
   "2900RS001A01F02.DI.AEN" : Bool AT %DB5014.DBX7.4, 500 ms
   "2900RS001A01F02.DI.AL_SUPR" : Bool AT %DB5014.DBX7.5, 500 ms
   "2900RS001A01F02.Q.PV_NORM" : Real AT %DB5014.DBD8, 500 ms
   "2900RS001A01F02.Q.PV_SCAL" : Real AT %DB5014.DBD12, 500 ms
   "2900RS001A01F02.ParentInfo" : TextRef, internal   // Имя родителя для попап окна, вкладка инфо. При експорте из ECS через скрипт заполняется автоматически, если теги копируются в ручную то требуется в ручную задатать свойство Start Value

HMI tags "2900RS001A01F03"
   "2900RS001A01F03.MSW" : 52809b66-421d-457f-8884-6f7a49d4e247 AT %DB5015.DBX18.0, 500 ms
   "2900RS001A01F03.DefaultText" : TextRef, internal   // Заголовок POPUP окна. При експорте из ECS через скрипт заполняется автоматически, если теги копируются в ручную то требуется в ручную задатать свойство Start Value
   "2900RS001A01F03.BlockInfo" : Array [0..2] of Int AT %DB5015.DBX38.0, 500 ms
   "2900RS001A01F03.StatusWork" : Int AT %DB5015.DBW242, 500 ms
   "2900RS001A01F03.FP_PARAM.DampingTime" : Int AT %DB5015.DBW50, 500 ms
   "2900RS001A01F03.FP_PARAM.Force_Value" : Real AT %DB5015.DBD52, 500 ms
   "2900RS001A01F03.FP_PARAM.Scale_Min" : Real AT %DB5015.DBD56, 500 ms
   "2900RS001A01F03.FP_PARAM.Scale_Max" : Real AT %DB5015.DBD60, 500 ms
   "2900RS001A01F03.FP_PARAM.Gradient" : Real AT %DB5015.DBD64, 500 ms
   "2900RS001A01F03.FP_PARAM.Grad_Pos" : Real AT %DB5015.DBD68, 500 ms
   "2900RS001A01F03.FP_PARAM.Grad_Neg" : Real AT %DB5015.DBD72, 500 ms
   "2900RS001A01F03.FP_PARAM.Grad_X" : Real AT %DB5015.DBD76, 500 ms
   "2900RS001A01F03.FP_PARAM.Gradient_Time_Pre" : Int AT %DB5015.DBW80, 500 ms
   "2900RS001A01F03.FP_PARAM.Gradient_Time_ACC" : Int AT %DB5015.DBW82, 500 ms
   "2900RS001A01F03.FP_PARAM.Alarm_Hyst" : Real AT %DB5015.DBD84, 500 ms
   "2900RS001A01F03.FP_PARAM.AlarmLimit_H3" : Real AT %DB5015.DBD88, 500 ms
   "2900RS001A01F03.FP_PARAM.AlarmLimit_H2" : Real AT %DB5015.DBD92, 500 ms
   "2900RS001A01F03.FP_PARAM.AlarmLimit_H1" : Real AT %DB5015.DBD96, 500 ms
   "2900RS001A01F03.FP_PARAM.AlarmLimit_L1" : Real AT %DB5015.DBD100, 500 ms
   "2900RS001A01F03.FP_PARAM.AlarmLimit_L2" : Real AT %DB5015.DBD104, 500 ms
   "2900RS001A01F03.FP_PARAM.AlarmLimit_L3" : Real AT %DB5015.DBD108, 500 ms
   "2900RS001A01F03.FP_PARAM.AlarmDelay_H3_Pre" : Int AT %DB5015.DBW112, 500 ms
   "2900RS001A01F03.FP_PARAM.AlarmDelay_H3_Acc" : Int AT %DB5015.DBW114, 500 ms
   "2900RS001A01F03.FP_PARAM.AlarmDelay_H2_Pre" : Int AT %DB5015.DBW116, 500 ms
   "2900RS001A01F03.FP_PARAM.AlarmDelay_H2_Acc" : Int AT %DB5015.DBW118, 500 ms
   "2900RS001A01F03.FP_PARAM.AlarmDelay_H1_Pre" : Int AT %DB5015.DBW120, 500 ms
   "2900RS001A01F03.FP_PARAM.AlarmDelay_H1_Acc" : Int AT %DB5015.DBW122, 500 ms
   "2900RS001A01F03.FP_PARAM.AlarmDelay_L1_Pre" : Int AT %DB5015.DBW124, 500 ms
   "2900RS001A01F03.FP_PARAM.AlarmDelay_L1_Acc" : Int AT %DB5015.DBW126, 500 ms
   "2900RS001A01F03.FP_PARAM.AlarmDelay_L2_Pre" : Int AT %DB5015.DBW128, 500 ms
   "2900RS001A01F03.FP_PARAM.AlarmDelay_L2_Acc" : Int AT %DB5015.DBW130, 500 ms
   "2900RS001A01F03.FP_PARAM.AlarmDelay_L3_Pre" : Int AT %DB5015.DBW132, 500 ms
   "2900RS001A01F03.FP_PARAM.AlarmDelay_L3_Acc" : Int AT %DB5015.DBW134, 500 ms
   "2900RS001A01F03.FP_PARAM.OpenLoopDelay_Pre" : Int AT %DB5015.DBW136, 500 ms
   "2900RS001A01F03.FP_PARAM.OpenLoopDelay_Acc" : Int AT %DB5015.DBW138, 500 ms
   "2900RS001A01F03.FP_PARAM.OverRangeDelay_Pre" : Int AT %DB5015.DBW140, 500 ms
   "2900RS001A01F03.FP_PARAM.OverRangeDelay_Acc" : Int AT %DB5015.DBW142, 500 ms
   "2900RS001A01F03.FP_PARAM.AuxLimit_H2_Value" : Real AT %DB5015.DBD144, 500 ms
   "2900RS001A01F03.FP_PARAM.AuxLimit_H1_Value" : Real AT %DB5015.DBD148, 500 ms
   "2900RS001A01F03.FP_PARAM.AuxLimit_L2_Value" : Real AT %DB5015.DBD152, 500 ms
   "2900RS001A01F03.FP_PARAM.AuxLimit_L1_Value" : Real AT %DB5015.DBD156, 500 ms
   "2900RS001A01F03.Unit" : TextRef, internal   // Еденицы измерения При експорте из ECS через скрипт заполняется автоматически, если теги копируются в ручную то требуется задатать свойство Text
   "2900RS001A01F03.Decimals" : TextRef, internal   // Формат отображения При експорте из ECS через скрипт, заполняется автоматически. Если теги копируются в ручную то требуется задатать свойство Text s999999.9
   "2900RS001A01F03.FP_EN.Square" : Bool AT %DB5015.DBX46.0, 500 ms
   "2900RS001A01F03.FP_EN.SquareRoot" : Bool AT %DB5015.DBX46.1, 500 ms
   "2900RS001A01F03.FP_EN.ParentSupress" : Bool AT %DB5015.DBX46.2, 500 ms
   "2900RS001A01F03.FP_EN.ParentSupressUnit" : Bool AT %DB5015.DBX46.3, 500 ms
   "2900RS001A01F03.FP_EN.Force" : Bool AT %DB5015.DBX46.4, 500 ms
   "2900RS001A01F03.FP_EN.Damping" : Bool AT %DB5015.DBX46.5, 500 ms
   "2900RS001A01F03.FP_EN.Gradient_Pos" : Bool AT %DB5015.DBX46.6, 500 ms
   "2900RS001A01F03.FP_EN.Gradient_Neg" : Bool AT %DB5015.DBX46.7, 500 ms
   "2900RS001A01F03.FP_EN.Hysteresis" : Bool AT %DB5015.DBX47.0, 500 ms
   "2900RS001A01F03.FP_EN.Alarm_H3" : Bool AT %DB5015.DBX47.1, 500 ms
   "2900RS001A01F03.FP_EN.Alarm_H2" : Bool AT %DB5015.DBX47.2, 500 ms
   "2900RS001A01F03.FP_EN.Alarm_H1" : Bool AT %DB5015.DBX47.3, 500 ms
   "2900RS001A01F03.FP_EN.Alarm_L1" : Bool AT %DB5015.DBX47.4, 500 ms
   "2900RS001A01F03.FP_EN.Alarm_L2" : Bool AT %DB5015.DBX47.5, 500 ms
   "2900RS001A01F03.FP_EN.Alarm_L3" : Bool AT %DB5015.DBX47.6, 500 ms
   "2900RS001A01F03.FP_EN.AlarmDelay_H3" : Bool AT %DB5015.DBX47.7, 500 ms
   "2900RS001A01F03.FP_EN.AlarmDelay_H2" : Bool AT %DB5015.DBX48.0, 500 ms
   "2900RS001A01F03.FP_EN.AlarmDelay_H1" : Bool AT %DB5015.DBX48.1, 500 ms
   "2900RS001A01F03.FP_EN.AlarmDelay_L1" : Bool AT %DB5015.DBX48.2, 500 ms
   "2900RS001A01F03.FP_EN.AlarmDelay_L2" : Bool AT %DB5015.DBX48.3, 500 ms
   "2900RS001A01F03.FP_EN.AlarmDelay_L3" : Bool AT %DB5015.DBX48.4, 500 ms
   "2900RS001A01F03.FP_EN.ROC_Warn" : Bool AT %DB5015.DBX48.5, 500 ms
   "2900RS001A01F03.FP_EN.U_Range_Warn" : Bool AT %DB5015.DBX48.6, 500 ms
   "2900RS001A01F03.FP_EN.O_Range_Warn" : Bool AT %DB5015.DBX48.7, 500 ms
   "2900RS001A01F03.trend_tag_name" : TextRef, internal   // Еденицы измерения При експорте из ECS через скрипт - заполняется автоматически, если теги копируются в ручную то требуется задатать свойство Text - имя тега для тренда
   "2900RS001A01F03.DQ.AL_H3" : Bool AT %DB5015.DBX16.0, 500 ms
   "2900RS001A01F03.DQ.AL_H2" : Bool AT %DB5015.DBX16.1, 500 ms
   "2900RS001A01F03.DQ.AL_H1" : Bool AT %DB5015.DBX16.2, 500 ms
   "2900RS001A01F03.DQ.AL_L1" : Bool AT %DB5015.DBX16.3, 500 ms
   "2900RS001A01F03.DQ.AL_L2" : Bool AT %DB5015.DBX16.4, 500 ms
   "2900RS001A01F03.DQ.AL_L3" : Bool AT %DB5015.DBX16.5, 500 ms
   "2900RS001A01F03.DQ.SIG_OK" : Bool AT %DB5015.DBX16.6, 500 ms
   "2900RS001A01F03.DQ.LIM_H2" : Bool AT %DB5015.DBX16.7, 500 ms
   "2900RS001A01F03.DQ.LIM_H1" : Bool AT %DB5015.DBX17.0, 500 ms
   "2900RS001A01F03.DQ.LIM_L1" : Bool AT %DB5015.DBX17.1, 500 ms
   "2900RS001A01F03.DQ.LIM_L2" : Bool AT %DB5015.DBX17.2, 500 ms
   "2900RS001A01F03.DQ.GR_P" : Bool AT %DB5015.DBX17.3, 500 ms
   "2900RS001A01F03.DQ.GR_N" : Bool AT %DB5015.DBX17.4, 500 ms
   "2900RS001A01F03.I.IN" : Real AT %DB5015.DBD2, 500 ms
   "2900RS001A01F03.I.SIG_TYPE" : Int AT %DB5015.DBW0, 500 ms
   "2900RS001A01F03.I.FI_BUS" : Byte AT %DB5015.DBB6, 500 ms
   "2900RS001A01F03.DI.U_RANGE" : Bool AT %DB5015.DBX7.0, 500 ms
   "2900RS001A01F03.DI.O_RANGE" : Bool AT %DB5015.DBX7.1, 500 ms
   "2900RS001A01F03.DI.SIG_FAULT" : Bool AT %DB5015.DBX7.2, 500 ms
   "2900RS001A01F03.DI.EnConfig" : Bool AT %DB5015.DBX7.3, 500 ms
   "2900RS001A01F03.DI.AEN" : Bool AT %DB5015.DBX7.4, 500 ms
   "2900RS001A01F03.DI.AL_SUPR" : Bool AT %DB5015.DBX7.5, 500 ms
   "2900RS001A01F03.Q.PV_NORM" : Real AT %DB5015.DBD8, 500 ms
   "2900RS001A01F03.Q.PV_SCAL" : Real AT %DB5015.DBD12, 500 ms
   "2900RS001A01F03.ParentInfo" : TextRef, internal   // Имя родителя для попап окна, вкладка инфо. При експорте из ECS через скрипт заполняется автоматически, если теги копируются в ручную то требуется в ручную задатать свойство Start Value

HMI tags "2900RS001A01F04"
   "2900RS001A01F04.MSW" : 52809b66-421d-457f-8884-6f7a49d4e247 AT %DB5016.DBX18.0, 500 ms
   "2900RS001A01F04.DefaultText" : TextRef, internal   // Заголовок POPUP окна. При експорте из ECS через скрипт заполняется автоматически, если теги копируются в ручную то требуется в ручную задатать свойство Start Value
   "2900RS001A01F04.BlockInfo" : Array [0..2] of Int AT %DB5016.DBX38.0, 500 ms
   "2900RS001A01F04.StatusWork" : Int AT %DB5016.DBW242, 500 ms
   "2900RS001A01F04.FP_PARAM.DampingTime" : Int AT %DB5016.DBW50, 500 ms
   "2900RS001A01F04.FP_PARAM.Force_Value" : Real AT %DB5016.DBD52, 500 ms
   "2900RS001A01F04.FP_PARAM.Scale_Min" : Real AT %DB5016.DBD56, 500 ms
   "2900RS001A01F04.FP_PARAM.Scale_Max" : Real AT %DB5016.DBD60, 500 ms
   "2900RS001A01F04.FP_PARAM.Gradient" : Real AT %DB5016.DBD64, 500 ms
   "2900RS001A01F04.FP_PARAM.Grad_Pos" : Real AT %DB5016.DBD68, 500 ms
   "2900RS001A01F04.FP_PARAM.Grad_Neg" : Real AT %DB5016.DBD72, 500 ms
   "2900RS001A01F04.FP_PARAM.Grad_X" : Real AT %DB5016.DBD76, 500 ms
   "2900RS001A01F04.FP_PARAM.Gradient_Time_Pre" : Int AT %DB5016.DBW80, 500 ms
   "2900RS001A01F04.FP_PARAM.Gradient_Time_ACC" : Int AT %DB5016.DBW82, 500 ms
   "2900RS001A01F04.FP_PARAM.Alarm_Hyst" : Real AT %DB5016.DBD84, 500 ms
   "2900RS001A01F04.FP_PARAM.AlarmLimit_H3" : Real AT %DB5016.DBD88, 500 ms
   "2900RS001A01F04.FP_PARAM.AlarmLimit_H2" : Real AT %DB5016.DBD92, 500 ms
   "2900RS001A01F04.FP_PARAM.AlarmLimit_H1" : Real AT %DB5016.DBD96, 500 ms
   "2900RS001A01F04.FP_PARAM.AlarmLimit_L1" : Real AT %DB5016.DBD100, 500 ms
   "2900RS001A01F04.FP_PARAM.AlarmLimit_L2" : Real AT %DB5016.DBD104, 500 ms
   "2900RS001A01F04.FP_PARAM.AlarmLimit_L3" : Real AT %DB5016.DBD108, 500 ms
   "2900RS001A01F04.FP_PARAM.AlarmDelay_H3_Pre" : Int AT %DB5016.DBW112, 500 ms
   "2900RS001A01F04.FP_PARAM.AlarmDelay_H3_Acc" : Int AT %DB5016.DBW114, 500 ms
   "2900RS001A01F04.FP_PARAM.AlarmDelay_H2_Pre" : Int AT %DB5016.DBW116, 500 ms
   "2900RS001A01F04.FP_PARAM.AlarmDelay_H2_Acc" : Int AT %DB5016.DBW118, 500 ms
   "2900RS001A01F04.FP_PARAM.AlarmDelay_H1_Pre" : Int AT %DB5016.DBW120, 500 ms
   "2900RS001A01F04.FP_PARAM.AlarmDelay_H1_Acc" : Int AT %DB5016.DBW122, 500 ms
   "2900RS001A01F04.FP_PARAM.AlarmDelay_L1_Pre" : Int AT %DB5016.DBW124, 500 ms
   "2900RS001A01F04.FP_PARAM.AlarmDelay_L1_Acc" : Int AT %DB5016.DBW126, 500 ms
   "2900RS001A01F04.FP_PARAM.AlarmDelay_L2_Pre" : Int AT %DB5016.DBW128, 500 ms
   "2900RS001A01F04.FP_PARAM.AlarmDelay_L2_Acc" : Int AT %DB5016.DBW130, 500 ms
   "2900RS001A01F04.FP_PARAM.AlarmDelay_L3_Pre" : Int AT %DB5016.DBW132, 500 ms
   "2900RS001A01F04.FP_PARAM.AlarmDelay_L3_Acc" : Int AT %DB5016.DBW134, 500 ms
   "2900RS001A01F04.FP_PARAM.OpenLoopDelay_Pre" : Int AT %DB5016.DBW136, 500 ms
   "2900RS001A01F04.FP_PARAM.OpenLoopDelay_Acc" : Int AT %DB5016.DBW138, 500 ms
   "2900RS001A01F04.FP_PARAM.OverRangeDelay_Pre" : Int AT %DB5016.DBW140, 500 ms
   "2900RS001A01F04.FP_PARAM.OverRangeDelay_Acc" : Int AT %DB5016.DBW142, 500 ms
   "2900RS001A01F04.FP_PARAM.AuxLimit_H2_Value" : Real AT %DB5016.DBD144, 500 ms
   "2900RS001A01F04.FP_PARAM.AuxLimit_H1_Value" : Real AT %DB5016.DBD148, 500 ms
   "2900RS001A01F04.FP_PARAM.AuxLimit_L2_Value" : Real AT %DB5016.DBD152, 500 ms
   "2900RS001A01F04.FP_PARAM.AuxLimit_L1_Value" : Real AT %DB5016.DBD156, 500 ms
   "2900RS001A01F04.Unit" : TextRef, internal   // Еденицы измерения При експорте из ECS через скрипт заполняется автоматически, если теги копируются в ручную то требуется задатать свойство Text
   "2900RS001A01F04.Decimals" : TextRef, internal   // Формат отображения При експорте из ECS через скрипт, заполняется автоматически. Если теги копируются в ручную то требуется задатать свойство Text s999999.9
   "2900RS001A01F04.FP_EN.Square" : Bool AT %DB5016.DBX46.0, 500 ms
   "2900RS001A01F04.FP_EN.SquareRoot" : Bool AT %DB5016.DBX46.1, 500 ms
   "2900RS001A01F04.FP_EN.ParentSupress" : Bool AT %DB5016.DBX46.2, 500 ms
   "2900RS001A01F04.FP_EN.ParentSupressUnit" : Bool AT %DB5016.DBX46.3, 500 ms
   "2900RS001A01F04.FP_EN.Force" : Bool AT %DB5016.DBX46.4, 500 ms
   "2900RS001A01F04.FP_EN.Damping" : Bool AT %DB5016.DBX46.5, 500 ms
   "2900RS001A01F04.FP_EN.Gradient_Pos" : Bool AT %DB5016.DBX46.6, 500 ms
   "2900RS001A01F04.FP_EN.Gradient_Neg" : Bool AT %DB5016.DBX46.7, 500 ms
   "2900RS001A01F04.FP_EN.Hysteresis" : Bool AT %DB5016.DBX47.0, 500 ms
   "2900RS001A01F04.FP_EN.Alarm_H3" : Bool AT %DB5016.DBX47.1, 500 ms
   "2900RS001A01F04.FP_EN.Alarm_H2" : Bool AT %DB5016.DBX47.2, 500 ms
   "2900RS001A01F04.FP_EN.Alarm_H1" : Bool AT %DB5016.DBX47.3, 500 ms
   "2900RS001A01F04.FP_EN.Alarm_L1" : Bool AT %DB5016.DBX47.4, 500 ms
   "2900RS001A01F04.FP_EN.Alarm_L2" : Bool AT %DB5016.DBX47.5, 500 ms
   "2900RS001A01F04.FP_EN.Alarm_L3" : Bool AT %DB5016.DBX47.6, 500 ms
   "2900RS001A01F04.FP_EN.AlarmDelay_H3" : Bool AT %DB5016.DBX47.7, 500 ms
   "2900RS001A01F04.FP_EN.AlarmDelay_H2" : Bool AT %DB5016.DBX48.0, 500 ms
   "2900RS001A01F04.FP_EN.AlarmDelay_H1" : Bool AT %DB5016.DBX48.1, 500 ms
   "2900RS001A01F04.FP_EN.AlarmDelay_L1" : Bool AT %DB5016.DBX48.2, 500 ms
   "2900RS001A01F04.FP_EN.AlarmDelay_L2" : Bool AT %DB5016.DBX48.3, 500 ms
   "2900RS001A01F04.FP_EN.AlarmDelay_L3" : Bool AT %DB5016.DBX48.4, 500 ms
   "2900RS001A01F04.FP_EN.ROC_Warn" : Bool AT %DB5016.DBX48.5, 500 ms
   "2900RS001A01F04.FP_EN.U_Range_Warn" : Bool AT %DB5016.DBX48.6, 500 ms
   "2900RS001A01F04.FP_EN.O_Range_Warn" : Bool AT %DB5016.DBX48.7, 500 ms
   "2900RS001A01F04.trend_tag_name" : TextRef, internal   // Еденицы измерения При експорте из ECS через скрипт - заполняется автоматически, если теги копируются в ручную то требуется задатать свойство Text - имя тега для тренда
   "2900RS001A01F04.DQ.AL_H3" : Bool AT %DB5016.DBX16.0, 500 ms
   "2900RS001A01F04.DQ.AL_H2" : Bool AT %DB5016.DBX16.1, 500 ms
   "2900RS001A01F04.DQ.AL_H1" : Bool AT %DB5016.DBX16.2, 500 ms
   "2900RS001A01F04.DQ.AL_L1" : Bool AT %DB5016.DBX16.3, 500 ms
   "2900RS001A01F04.DQ.AL_L2" : Bool AT %DB5016.DBX16.4, 500 ms
   "2900RS001A01F04.DQ.AL_L3" : Bool AT %DB5016.DBX16.5, 500 ms
   "2900RS001A01F04.DQ.SIG_OK" : Bool AT %DB5016.DBX16.6, 500 ms
   "2900RS001A01F04.DQ.LIM_H2" : Bool AT %DB5016.DBX16.7, 500 ms
   "2900RS001A01F04.DQ.LIM_H1" : Bool AT %DB5016.DBX17.0, 500 ms
   "2900RS001A01F04.DQ.LIM_L1" : Bool AT %DB5016.DBX17.1, 500 ms
   "2900RS001A01F04.DQ.LIM_L2" : Bool AT %DB5016.DBX17.2, 500 ms
   "2900RS001A01F04.DQ.GR_P" : Bool AT %DB5016.DBX17.3, 500 ms
   "2900RS001A01F04.DQ.GR_N" : Bool AT %DB5016.DBX17.4, 500 ms
   "2900RS001A01F04.I.IN" : Real AT %DB5016.DBD2, 500 ms
   "2900RS001A01F04.I.SIG_TYPE" : Int AT %DB5016.DBW0, 500 ms
   "2900RS001A01F04.I.FI_BUS" : Byte AT %DB5016.DBB6, 500 ms
   "2900RS001A01F04.DI.U_RANGE" : Bool AT %DB5016.DBX7.0, 500 ms
   "2900RS001A01F04.DI.O_RANGE" : Bool AT %DB5016.DBX7.1, 500 ms
   "2900RS001A01F04.DI.SIG_FAULT" : Bool AT %DB5016.DBX7.2, 500 ms
   "2900RS001A01F04.DI.EnConfig" : Bool AT %DB5016.DBX7.3, 500 ms
   "2900RS001A01F04.DI.AEN" : Bool AT %DB5016.DBX7.4, 500 ms
   "2900RS001A01F04.DI.AL_SUPR" : Bool AT %DB5016.DBX7.5, 500 ms
   "2900RS001A01F04.Q.PV_NORM" : Real AT %DB5016.DBD8, 500 ms
   "2900RS001A01F04.Q.PV_SCAL" : Real AT %DB5016.DBD12, 500 ms
   "2900RS001A01F04.ParentInfo" : TextRef, internal   // Имя родителя для попап окна, вкладка инфо. При експорте из ECS через скрипт заполняется автоматически, если теги копируются в ручную то требуется в ручную задатать свойство Start Value

HMI tags "2900RS001A01F05"
   "2900RS001A01F05.MSW" : 52809b66-421d-457f-8884-6f7a49d4e247 AT %DB5017.DBX18.0, 500 ms
   "2900RS001A01F05.DefaultText" : TextRef, internal   // Заголовок POPUP окна. При експорте из ECS через скрипт заполняется автоматически, если теги копируются в ручную то требуется в ручную задатать свойство Start Value
   "2900RS001A01F05.BlockInfo" : Array [0..2] of Int AT %DB5017.DBX38.0, 500 ms
   "2900RS001A01F05.StatusWork" : Int AT %DB5017.DBW242, 500 ms
   "2900RS001A01F05.FP_PARAM.DampingTime" : Int AT %DB5017.DBW50, 500 ms
   "2900RS001A01F05.FP_PARAM.Force_Value" : Real AT %DB5017.DBD52, 500 ms
   "2900RS001A01F05.FP_PARAM.Scale_Min" : Real AT %DB5017.DBD56, 500 ms
   "2900RS001A01F05.FP_PARAM.Scale_Max" : Real AT %DB5017.DBD60, 500 ms
   "2900RS001A01F05.FP_PARAM.Gradient" : Real AT %DB5017.DBD64, 500 ms
   "2900RS001A01F05.FP_PARAM.Grad_Pos" : Real AT %DB5017.DBD68, 500 ms
   "2900RS001A01F05.FP_PARAM.Grad_Neg" : Real AT %DB5017.DBD72, 500 ms
   "2900RS001A01F05.FP_PARAM.Grad_X" : Real AT %DB5017.DBD76, 500 ms
   "2900RS001A01F05.FP_PARAM.Gradient_Time_Pre" : Int AT %DB5017.DBW80, 500 ms
   "2900RS001A01F05.FP_PARAM.Gradient_Time_ACC" : Int AT %DB5017.DBW82, 500 ms
   "2900RS001A01F05.FP_PARAM.Alarm_Hyst" : Real AT %DB5017.DBD84, 500 ms
   "2900RS001A01F05.FP_PARAM.AlarmLimit_H3" : Real AT %DB5017.DBD88, 500 ms
   "2900RS001A01F05.FP_PARAM.AlarmLimit_H2" : Real AT %DB5017.DBD92, 500 ms
   "2900RS001A01F05.FP_PARAM.AlarmLimit_H1" : Real AT %DB5017.DBD96, 500 ms
   "2900RS001A01F05.FP_PARAM.AlarmLimit_L1" : Real AT %DB5017.DBD100, 500 ms
   "2900RS001A01F05.FP_PARAM.AlarmLimit_L2" : Real AT %DB5017.DBD104, 500 ms
   "2900RS001A01F05.FP_PARAM.AlarmLimit_L3" : Real AT %DB5017.DBD108, 500 ms
   "2900RS001A01F05.FP_PARAM.AlarmDelay_H3_Pre" : Int AT %DB5017.DBW112, 500 ms
   "2900RS001A01F05.FP_PARAM.AlarmDelay_H3_Acc" : Int AT %DB5017.DBW114, 500 ms
   "2900RS001A01F05.FP_PARAM.AlarmDelay_H2_Pre" : Int AT %DB5017.DBW116, 500 ms
   "2900RS001A01F05.FP_PARAM.AlarmDelay_H2_Acc" : Int AT %DB5017.DBW118, 500 ms
   "2900RS001A01F05.FP_PARAM.AlarmDelay_H1_Pre" : Int AT %DB5017.DBW120, 500 ms
   "2900RS001A01F05.FP_PARAM.AlarmDelay_H1_Acc" : Int AT %DB5017.DBW122, 500 ms
   "2900RS001A01F05.FP_PARAM.AlarmDelay_L1_Pre" : Int AT %DB5017.DBW124, 500 ms
   "2900RS001A01F05.FP_PARAM.AlarmDelay_L1_Acc" : Int AT %DB5017.DBW126, 500 ms
   "2900RS001A01F05.FP_PARAM.AlarmDelay_L2_Pre" : Int AT %DB5017.DBW128, 500 ms
   "2900RS001A01F05.FP_PARAM.AlarmDelay_L2_Acc" : Int AT %DB5017.DBW130, 500 ms
   "2900RS001A01F05.FP_PARAM.AlarmDelay_L3_Pre" : Int AT %DB5017.DBW132, 500 ms
   "2900RS001A01F05.FP_PARAM.AlarmDelay_L3_Acc" : Int AT %DB5017.DBW134, 500 ms
   "2900RS001A01F05.FP_PARAM.OpenLoopDelay_Pre" : Int AT %DB5017.DBW136, 500 ms
   "2900RS001A01F05.FP_PARAM.OpenLoopDelay_Acc" : Int AT %DB5017.DBW138, 500 ms
   "2900RS001A01F05.FP_PARAM.OverRangeDelay_Pre" : Int AT %DB5017.DBW140, 500 ms
   "2900RS001A01F05.FP_PARAM.OverRangeDelay_Acc" : Int AT %DB5017.DBW142, 500 ms
   "2900RS001A01F05.FP_PARAM.AuxLimit_H2_Value" : Real AT %DB5017.DBD144, 500 ms
   "2900RS001A01F05.FP_PARAM.AuxLimit_H1_Value" : Real AT %DB5017.DBD148, 500 ms
   "2900RS001A01F05.FP_PARAM.AuxLimit_L2_Value" : Real AT %DB5017.DBD152, 500 ms
   "2900RS001A01F05.FP_PARAM.AuxLimit_L1_Value" : Real AT %DB5017.DBD156, 500 ms
   "2900RS001A01F05.Unit" : TextRef, internal   // Еденицы измерения При експорте из ECS через скрипт заполняется автоматически, если теги копируются в ручную то требуется задатать свойство Text
   "2900RS001A01F05.Decimals" : TextRef, internal   // Формат отображения При експорте из ECS через скрипт, заполняется автоматически. Если теги копируются в ручную то требуется задатать свойство Text s999999.9
   "2900RS001A01F05.FP_EN.Square" : Bool AT %DB5017.DBX46.0, 500 ms
   "2900RS001A01F05.FP_EN.SquareRoot" : Bool AT %DB5017.DBX46.1, 500 ms
   "2900RS001A01F05.FP_EN.ParentSupress" : Bool AT %DB5017.DBX46.2, 500 ms
   "2900RS001A01F05.FP_EN.ParentSupressUnit" : Bool AT %DB5017.DBX46.3, 500 ms
   "2900RS001A01F05.FP_EN.Force" : Bool AT %DB5017.DBX46.4, 500 ms
   "2900RS001A01F05.FP_EN.Damping" : Bool AT %DB5017.DBX46.5, 500 ms
   "2900RS001A01F05.FP_EN.Gradient_Pos" : Bool AT %DB5017.DBX46.6, 500 ms
   "2900RS001A01F05.FP_EN.Gradient_Neg" : Bool AT %DB5017.DBX46.7, 500 ms
   "2900RS001A01F05.FP_EN.Hysteresis" : Bool AT %DB5017.DBX47.0, 500 ms
   "2900RS001A01F05.FP_EN.Alarm_H3" : Bool AT %DB5017.DBX47.1, 500 ms
   "2900RS001A01F05.FP_EN.Alarm_H2" : Bool AT %DB5017.DBX47.2, 500 ms
   "2900RS001A01F05.FP_EN.Alarm_H1" : Bool AT %DB5017.DBX47.3, 500 ms
   "2900RS001A01F05.FP_EN.Alarm_L1" : Bool AT %DB5017.DBX47.4, 500 ms
   "2900RS001A01F05.FP_EN.Alarm_L2" : Bool AT %DB5017.DBX47.5, 500 ms
   "2900RS001A01F05.FP_EN.Alarm_L3" : Bool AT %DB5017.DBX47.6, 500 ms
   "2900RS001A01F05.FP_EN.AlarmDelay_H3" : Bool AT %DB5017.DBX47.7, 500 ms
   "2900RS001A01F05.FP_EN.AlarmDelay_H2" : Bool AT %DB5017.DBX48.0, 500 ms
   "2900RS001A01F05.FP_EN.AlarmDelay_H1" : Bool AT %DB5017.DBX48.1, 500 ms
   "2900RS001A01F05.FP_EN.AlarmDelay_L1" : Bool AT %DB5017.DBX48.2, 500 ms
   "2900RS001A01F05.FP_EN.AlarmDelay_L2" : Bool AT %DB5017.DBX48.3, 500 ms
   "2900RS001A01F05.FP_EN.AlarmDelay_L3" : Bool AT %DB5017.DBX48.4, 500 ms
   "2900RS001A01F05.FP_EN.ROC_Warn" : Bool AT %DB5017.DBX48.5, 500 ms
   "2900RS001A01F05.FP_EN.U_Range_Warn" : Bool AT %DB5017.DBX48.6, 500 ms
   "2900RS001A01F05.FP_EN.O_Range_Warn" : Bool AT %DB5017.DBX48.7, 500 ms
   "2900RS001A01F05.trend_tag_name" : TextRef, internal   // Еденицы измерения При експорте из ECS через скрипт - заполняется автоматически, если теги копируются в ручную то требуется задатать свойство Text - имя тега для тренда
   "2900RS001A01F05.DQ.AL_H3" : Bool AT %DB5017.DBX16.0, 500 ms
   "2900RS001A01F05.DQ.AL_H2" : Bool AT %DB5017.DBX16.1, 500 ms
   "2900RS001A01F05.DQ.AL_H1" : Bool AT %DB5017.DBX16.2, 500 ms
   "2900RS001A01F05.DQ.AL_L1" : Bool AT %DB5017.DBX16.3, 500 ms
   "2900RS001A01F05.DQ.AL_L2" : Bool AT %DB5017.DBX16.4, 500 ms
   "2900RS001A01F05.DQ.AL_L3" : Bool AT %DB5017.DBX16.5, 500 ms
   "2900RS001A01F05.DQ.SIG_OK" : Bool AT %DB5017.DBX16.6, 500 ms
   "2900RS001A01F05.DQ.LIM_H2" : Bool AT %DB5017.DBX16.7, 500 ms
   "2900RS001A01F05.DQ.LIM_H1" : Bool AT %DB5017.DBX17.0, 500 ms
   "2900RS001A01F05.DQ.LIM_L1" : Bool AT %DB5017.DBX17.1, 500 ms
   "2900RS001A01F05.DQ.LIM_L2" : Bool AT %DB5017.DBX17.2, 500 ms
   "2900RS001A01F05.DQ.GR_P" : Bool AT %DB5017.DBX17.3, 500 ms
   "2900RS001A01F05.DQ.GR_N" : Bool AT %DB5017.DBX17.4, 500 ms
   "2900RS001A01F05.I.IN" : Real AT %DB5017.DBD2, 500 ms
   "2900RS001A01F05.I.SIG_TYPE" : Int AT %DB5017.DBW0, 500 ms
   "2900RS001A01F05.I.FI_BUS" : Byte AT %DB5017.DBB6, 500 ms
   "2900RS001A01F05.DI.U_RANGE" : Bool AT %DB5017.DBX7.0, 500 ms
   "2900RS001A01F05.DI.O_RANGE" : Bool AT %DB5017.DBX7.1, 500 ms
   "2900RS001A01F05.DI.SIG_FAULT" : Bool AT %DB5017.DBX7.2, 500 ms
   "2900RS001A01F05.DI.EnConfig" : Bool AT %DB5017.DBX7.3, 500 ms
   "2900RS001A01F05.DI.AEN" : Bool AT %DB5017.DBX7.4, 500 ms
   "2900RS001A01F05.DI.AL_SUPR" : Bool AT %DB5017.DBX7.5, 500 ms
   "2900RS001A01F05.Q.PV_NORM" : Real AT %DB5017.DBD8, 500 ms
   "2900RS001A01F05.Q.PV_SCAL" : Real AT %DB5017.DBD12, 500 ms
   "2900RS001A01F05.ParentInfo" : TextRef, internal   // Имя родителя для попап окна, вкладка инфо. При експорте из ECS через скрипт заполняется автоматически, если теги копируются в ручную то требуется в ручную задатать свойство Start Value

HMI tags "2900RS001A01F06"
   "2900RS001A01F06.MSW" : 52809b66-421d-457f-8884-6f7a49d4e247 AT %DB5018.DBX18.0, 500 ms
   "2900RS001A01F06.DefaultText" : TextRef, internal   // Заголовок POPUP окна. При експорте из ECS через скрипт заполняется автоматически, если теги копируются в ручную то требуется в ручную задатать свойство Start Value
   "2900RS001A01F06.BlockInfo" : Array [0..2] of Int AT %DB5018.DBX38.0, 500 ms
   "2900RS001A01F06.StatusWork" : Int AT %DB5018.DBW242, 500 ms
   "2900RS001A01F06.FP_PARAM.DampingTime" : Int AT %DB5018.DBW50, 500 ms
   "2900RS001A01F06.FP_PARAM.Force_Value" : Real AT %DB5018.DBD52, 500 ms
   "2900RS001A01F06.FP_PARAM.Scale_Min" : Real AT %DB5018.DBD56, 500 ms
   "2900RS001A01F06.FP_PARAM.Scale_Max" : Real AT %DB5018.DBD60, 500 ms
   "2900RS001A01F06.FP_PARAM.Gradient" : Real AT %DB5018.DBD64, 500 ms
   "2900RS001A01F06.FP_PARAM.Grad_Pos" : Real AT %DB5018.DBD68, 500 ms
   "2900RS001A01F06.FP_PARAM.Grad_Neg" : Real AT %DB5018.DBD72, 500 ms
   "2900RS001A01F06.FP_PARAM.Grad_X" : Real AT %DB5018.DBD76, 500 ms
   "2900RS001A01F06.FP_PARAM.Gradient_Time_Pre" : Int AT %DB5018.DBW80, 500 ms
   "2900RS001A01F06.FP_PARAM.Gradient_Time_ACC" : Int AT %DB5018.DBW82, 500 ms
   "2900RS001A01F06.FP_PARAM.Alarm_Hyst" : Real AT %DB5018.DBD84, 500 ms
   "2900RS001A01F06.FP_PARAM.AlarmLimit_H3" : Real AT %DB5018.DBD88, 500 ms
   "2900RS001A01F06.FP_PARAM.AlarmLimit_H2" : Real AT %DB5018.DBD92, 500 ms
   "2900RS001A01F06.FP_PARAM.AlarmLimit_H1" : Real AT %DB5018.DBD96, 500 ms
   "2900RS001A01F06.FP_PARAM.AlarmLimit_L1" : Real AT %DB5018.DBD100, 500 ms
   "2900RS001A01F06.FP_PARAM.AlarmLimit_L2" : Real AT %DB5018.DBD104, 500 ms
   "2900RS001A01F06.FP_PARAM.AlarmLimit_L3" : Real AT %DB5018.DBD108, 500 ms
   "2900RS001A01F06.FP_PARAM.AlarmDelay_H3_Pre" : Int AT %DB5018.DBW112, 500 ms
   "2900RS001A01F06.FP_PARAM.AlarmDelay_H3_Acc" : Int AT %DB5018.DBW114, 500 ms
   "2900RS001A01F06.FP_PARAM.AlarmDelay_H2_Pre" : Int AT %DB5018.DBW116, 500 ms
   "2900RS001A01F06.FP_PARAM.AlarmDelay_H2_Acc" : Int AT %DB5018.DBW118, 500 ms
   "2900RS001A01F06.FP_PARAM.AlarmDelay_H1_Pre" : Int AT %DB5018.DBW120, 500 ms
   "2900RS001A01F06.FP_PARAM.AlarmDelay_H1_Acc" : Int AT %DB5018.DBW122, 500 ms
   "2900RS001A01F06.FP_PARAM.AlarmDelay_L1_Pre" : Int AT %DB5018.DBW124, 500 ms
   "2900RS001A01F06.FP_PARAM.AlarmDelay_L1_Acc" : Int AT %DB5018.DBW126, 500 ms
   "2900RS001A01F06.FP_PARAM.AlarmDelay_L2_Pre" : Int AT %DB5018.DBW128, 500 ms
   "2900RS001A01F06.FP_PARAM.AlarmDelay_L2_Acc" : Int AT %DB5018.DBW130, 500 ms
   "2900RS001A01F06.FP_PARAM.AlarmDelay_L3_Pre" : Int AT %DB5018.DBW132, 500 ms
   "2900RS001A01F06.FP_PARAM.AlarmDelay_L3_Acc" : Int AT %DB5018.DBW134, 500 ms
   "2900RS001A01F06.FP_PARAM.OpenLoopDelay_Pre" : Int AT %DB5018.DBW136, 500 ms
   "2900RS001A01F06.FP_PARAM.OpenLoopDelay_Acc" : Int AT %DB5018.DBW138, 500 ms
   "2900RS001A01F06.FP_PARAM.OverRangeDelay_Pre" : Int AT %DB5018.DBW140, 500 ms
   "2900RS001A01F06.FP_PARAM.OverRangeDelay_Acc" : Int AT %DB5018.DBW142, 500 ms
   "2900RS001A01F06.FP_PARAM.AuxLimit_H2_Value" : Real AT %DB5018.DBD144, 500 ms
   "2900RS001A01F06.FP_PARAM.AuxLimit_H1_Value" : Real AT %DB5018.DBD148, 500 ms
   "2900RS001A01F06.FP_PARAM.AuxLimit_L2_Value" : Real AT %DB5018.DBD152, 500 ms
   "2900RS001A01F06.FP_PARAM.AuxLimit_L1_Value" : Real AT %DB5018.DBD156, 500 ms
   "2900RS001A01F06.Unit" : TextRef, internal   // Еденицы измерения При експорте из ECS через скрипт заполняется автоматически, если теги копируются в ручную то требуется задатать свойство Text
   "2900RS001A01F06.Decimals" : TextRef, internal   // Формат отображения При експорте из ECS через скрипт, заполняется автоматически. Если теги копируются в ручную то требуется задатать свойство Text s999999.9
   "2900RS001A01F06.FP_EN.Square" : Bool AT %DB5018.DBX46.0, 500 ms
   "2900RS001A01F06.FP_EN.SquareRoot" : Bool AT %DB5018.DBX46.1, 500 ms
   "2900RS001A01F06.FP_EN.ParentSupress" : Bool AT %DB5018.DBX46.2, 500 ms
   "2900RS001A01F06.FP_EN.ParentSupressUnit" : Bool AT %DB5018.DBX46.3, 500 ms
   "2900RS001A01F06.FP_EN.Force" : Bool AT %DB5018.DBX46.4, 500 ms
   "2900RS001A01F06.FP_EN.Damping" : Bool AT %DB5018.DBX46.5, 500 ms
   "2900RS001A01F06.FP_EN.Gradient_Pos" : Bool AT %DB5018.DBX46.6, 500 ms
   "2900RS001A01F06.FP_EN.Gradient_Neg" : Bool AT %DB5018.DBX46.7, 500 ms
   "2900RS001A01F06.FP_EN.Hysteresis" : Bool AT %DB5018.DBX47.0, 500 ms
   "2900RS001A01F06.FP_EN.Alarm_H3" : Bool AT %DB5018.DBX47.1, 500 ms
   "2900RS001A01F06.FP_EN.Alarm_H2" : Bool AT %DB5018.DBX47.2, 500 ms
   "2900RS001A01F06.FP_EN.Alarm_H1" : Bool AT %DB5018.DBX47.3, 500 ms
   "2900RS001A01F06.FP_EN.Alarm_L1" : Bool AT %DB5018.DBX47.4, 500 ms
   "2900RS001A01F06.FP_EN.Alarm_L2" : Bool AT %DB5018.DBX47.5, 500 ms
   "2900RS001A01F06.FP_EN.Alarm_L3" : Bool AT %DB5018.DBX47.6, 500 ms
   "2900RS001A01F06.FP_EN.AlarmDelay_H3" : Bool AT %DB5018.DBX47.7, 500 ms
   "2900RS001A01F06.FP_EN.AlarmDelay_H2" : Bool AT %DB5018.DBX48.0, 500 ms
   "2900RS001A01F06.FP_EN.AlarmDelay_H1" : Bool AT %DB5018.DBX48.1, 500 ms
   "2900RS001A01F06.FP_EN.AlarmDelay_L1" : Bool AT %DB5018.DBX48.2, 500 ms
   "2900RS001A01F06.FP_EN.AlarmDelay_L2" : Bool AT %DB5018.DBX48.3, 500 ms
   "2900RS001A01F06.FP_EN.AlarmDelay_L3" : Bool AT %DB5018.DBX48.4, 500 ms
   "2900RS001A01F06.FP_EN.ROC_Warn" : Bool AT %DB5018.DBX48.5, 500 ms
   "2900RS001A01F06.FP_EN.U_Range_Warn" : Bool AT %DB5018.DBX48.6, 500 ms
   "2900RS001A01F06.FP_EN.O_Range_Warn" : Bool AT %DB5018.DBX48.7, 500 ms
   "2900RS001A01F06.trend_tag_name" : TextRef, internal   // Еденицы измерения При експорте из ECS через скрипт - заполняется автоматически, если теги копируются в ручную то требуется задатать свойство Text - имя тега для тренда
   "2900RS001A01F06.DQ.AL_H3" : Bool AT %DB5018.DBX16.0, 500 ms
   "2900RS001A01F06.DQ.AL_H2" : Bool AT %DB5018.DBX16.1, 500 ms
   "2900RS001A01F06.DQ.AL_H1" : Bool AT %DB5018.DBX16.2, 500 ms
   "2900RS001A01F06.DQ.AL_L1" : Bool AT %DB5018.DBX16.3, 500 ms
   "2900RS001A01F06.DQ.AL_L2" : Bool AT %DB5018.DBX16.4, 500 ms
   "2900RS001A01F06.DQ.AL_L3" : Bool AT %DB5018.DBX16.5, 500 ms
   "2900RS001A01F06.DQ.SIG_OK" : Bool AT %DB5018.DBX16.6, 500 ms
   "2900RS001A01F06.DQ.LIM_H2" : Bool AT %DB5018.DBX16.7, 500 ms
   "2900RS001A01F06.DQ.LIM_H1" : Bool AT %DB5018.DBX17.0, 500 ms
   "2900RS001A01F06.DQ.LIM_L1" : Bool AT %DB5018.DBX17.1, 500 ms
   "2900RS001A01F06.DQ.LIM_L2" : Bool AT %DB5018.DBX17.2, 500 ms
   "2900RS001A01F06.DQ.GR_P" : Bool AT %DB5018.DBX17.3, 500 ms
   "2900RS001A01F06.DQ.GR_N" : Bool AT %DB5018.DBX17.4, 500 ms
   "2900RS001A01F06.I.IN" : Real AT %DB5018.DBD2, 500 ms
   "2900RS001A01F06.I.SIG_TYPE" : Int AT %DB5018.DBW0, 500 ms
   "2900RS001A01F06.I.FI_BUS" : Byte AT %DB5018.DBB6, 500 ms
   "2900RS001A01F06.DI.U_RANGE" : Bool AT %DB5018.DBX7.0, 500 ms
   "2900RS001A01F06.DI.O_RANGE" : Bool AT %DB5018.DBX7.1, 500 ms
   "2900RS001A01F06.DI.SIG_FAULT" : Bool AT %DB5018.DBX7.2, 500 ms
   "2900RS001A01F06.DI.EnConfig" : Bool AT %DB5018.DBX7.3, 500 ms
   "2900RS001A01F06.DI.AEN" : Bool AT %DB5018.DBX7.4, 500 ms
   "2900RS001A01F06.DI.AL_SUPR" : Bool AT %DB5018.DBX7.5, 500 ms
   "2900RS001A01F06.Q.PV_NORM" : Real AT %DB5018.DBD8, 500 ms
   "2900RS001A01F06.Q.PV_SCAL" : Real AT %DB5018.DBD12, 500 ms
   "2900RS001A01F06.ParentInfo" : TextRef, internal   // Имя родителя для попап окна, вкладка инфо. При експорте из ECS через скрипт заполняется автоматически, если теги копируются в ручную то требуется в ручную задатать свойство Start Value

HMI tags "2900RS001A01L01"
   "2900RS001A01L01.MSW" : 52809b66-421d-457f-8884-6f7a49d4e247 AT %DB5019.DBX18.0, 500 ms
   "2900RS001A01L01.DefaultText" : TextRef, internal   // Заголовок POPUP окна. При експорте из ECS через скрипт заполняется автоматически, если теги копируются в ручную то требуется в ручную задатать свойство Start Value
   "2900RS001A01L01.BlockInfo" : Array [0..2] of Int AT %DB5019.DBX38.0, 500 ms
   "2900RS001A01L01.StatusWork" : Int AT %DB5019.DBW242, 500 ms
   "2900RS001A01L01.FP_PARAM.DampingTime" : Int AT %DB5019.DBW50, 500 ms
   "2900RS001A01L01.FP_PARAM.Force_Value" : Real AT %DB5019.DBD52, 500 ms
   "2900RS001A01L01.FP_PARAM.Scale_Min" : Real AT %DB5019.DBD56, 500 ms
   "2900RS001A01L01.FP_PARAM.Scale_Max" : Real AT %DB5019.DBD60, 500 ms
   "2900RS001A01L01.FP_PARAM.Gradient" : Real AT %DB5019.DBD64, 500 ms
   "2900RS001A01L01.FP_PARAM.Grad_Pos" : Real AT %DB5019.DBD68, 500 ms
   "2900RS001A01L01.FP_PARAM.Grad_Neg" : Real AT %DB5019.DBD72, 500 ms
   "2900RS001A01L01.FP_PARAM.Grad_X" : Real AT %DB5019.DBD76, 500 ms
   "2900RS001A01L01.FP_PARAM.Gradient_Time_Pre" : Int AT %DB5019.DBW80, 500 ms
   "2900RS001A01L01.FP_PARAM.Gradient_Time_ACC" : Int AT %DB5019.DBW82, 500 ms
   "2900RS001A01L01.FP_PARAM.Alarm_Hyst" : Real AT %DB5019.DBD84, 500 ms
   "2900RS001A01L01.FP_PARAM.AlarmLimit_H3" : Real AT %DB5019.DBD88, 500 ms
   "2900RS001A01L01.FP_PARAM.AlarmLimit_H2" : Real AT %DB5019.DBD92, 500 ms
   "2900RS001A01L01.FP_PARAM.AlarmLimit_H1" : Real AT %DB5019.DBD96, 500 ms
   "2900RS001A01L01.FP_PARAM.AlarmLimit_L1" : Real AT %DB5019.DBD100, 500 ms
   "2900RS001A01L01.FP_PARAM.AlarmLimit_L2" : Real AT %DB5019.DBD104, 500 ms
   "2900RS001A01L01.FP_PARAM.AlarmLimit_L3" : Real AT %DB5019.DBD108, 500 ms
   "2900RS001A01L01.FP_PARAM.AlarmDelay_H3_Pre" : Int AT %DB5019.DBW112, 500 ms
   "2900RS001A01L01.FP_PARAM.AlarmDelay_H3_Acc" : Int AT %DB5019.DBW114, 500 ms
   "2900RS001A01L01.FP_PARAM.AlarmDelay_H2_Pre" : Int AT %DB5019.DBW116, 500 ms
   "2900RS001A01L01.FP_PARAM.AlarmDelay_H2_Acc" : Int AT %DB5019.DBW118, 500 ms
   "2900RS001A01L01.FP_PARAM.AlarmDelay_H1_Pre" : Int AT %DB5019.DBW120, 500 ms
   "2900RS001A01L01.FP_PARAM.AlarmDelay_H1_Acc" : Int AT %DB5019.DBW122, 500 ms
   "2900RS001A01L01.FP_PARAM.AlarmDelay_L1_Pre" : Int AT %DB5019.DBW124, 500 ms
   "2900RS001A01L01.FP_PARAM.AlarmDelay_L1_Acc" : Int AT %DB5019.DBW126, 500 ms
   "2900RS001A01L01.FP_PARAM.AlarmDelay_L2_Pre" : Int AT %DB5019.DBW128, 500 ms
   "2900RS001A01L01.FP_PARAM.AlarmDelay_L2_Acc" : Int AT %DB5019.DBW130, 500 ms
   "2900RS001A01L01.FP_PARAM.AlarmDelay_L3_Pre" : Int AT %DB5019.DBW132, 500 ms
   "2900RS001A01L01.FP_PARAM.AlarmDelay_L3_Acc" : Int AT %DB5019.DBW134, 500 ms
   "2900RS001A01L01.FP_PARAM.OpenLoopDelay_Pre" : Int AT %DB5019.DBW136, 500 ms
   "2900RS001A01L01.FP_PARAM.OpenLoopDelay_Acc" : Int AT %DB5019.DBW138, 500 ms
   "2900RS001A01L01.FP_PARAM.OverRangeDelay_Pre" : Int AT %DB5019.DBW140, 500 ms
   "2900RS001A01L01.FP_PARAM.OverRangeDelay_Acc" : Int AT %DB5019.DBW142, 500 ms
   "2900RS001A01L01.FP_PARAM.AuxLimit_H2_Value" : Real AT %DB5019.DBD144, 500 ms
   "2900RS001A01L01.FP_PARAM.AuxLimit_H1_Value" : Real AT %DB5019.DBD148, 500 ms
   "2900RS001A01L01.FP_PARAM.AuxLimit_L2_Value" : Real AT %DB5019.DBD152, 500 ms
   "2900RS001A01L01.FP_PARAM.AuxLimit_L1_Value" : Real AT %DB5019.DBD156, 500 ms
   "2900RS001A01L01.Unit" : TextRef, internal   // Еденицы измерения При експорте из ECS через скрипт заполняется автоматически, если теги копируются в ручную то требуется задатать свойство Text
   "2900RS001A01L01.Decimals" : TextRef, internal   // Формат отображения При експорте из ECS через скрипт, заполняется автоматически. Если теги копируются в ручную то требуется задатать свойство Text s999999.9
   "2900RS001A01L01.FP_EN.Square" : Bool AT %DB5019.DBX46.0, 500 ms
   "2900RS001A01L01.FP_EN.SquareRoot" : Bool AT %DB5019.DBX46.1, 500 ms
   "2900RS001A01L01.FP_EN.ParentSupress" : Bool AT %DB5019.DBX46.2, 500 ms
   "2900RS001A01L01.FP_EN.ParentSupressUnit" : Bool AT %DB5019.DBX46.3, 500 ms
   "2900RS001A01L01.FP_EN.Force" : Bool AT %DB5019.DBX46.4, 500 ms
   "2900RS001A01L01.FP_EN.Damping" : Bool AT %DB5019.DBX46.5, 500 ms
   "2900RS001A01L01.FP_EN.Gradient_Pos" : Bool AT %DB5019.DBX46.6, 500 ms
   "2900RS001A01L01.FP_EN.Gradient_Neg" : Bool AT %DB5019.DBX46.7, 500 ms
   "2900RS001A01L01.FP_EN.Hysteresis" : Bool AT %DB5019.DBX47.0, 500 ms
   "2900RS001A01L01.FP_EN.Alarm_H3" : Bool AT %DB5019.DBX47.1, 500 ms
   "2900RS001A01L01.FP_EN.Alarm_H2" : Bool AT %DB5019.DBX47.2, 500 ms
   "2900RS001A01L01.FP_EN.Alarm_H1" : Bool AT %DB5019.DBX47.3, 500 ms
   "2900RS001A01L01.FP_EN.Alarm_L1" : Bool AT %DB5019.DBX47.4, 500 ms
   "2900RS001A01L01.FP_EN.Alarm_L2" : Bool AT %DB5019.DBX47.5, 500 ms
   "2900RS001A01L01.FP_EN.Alarm_L3" : Bool AT %DB5019.DBX47.6, 500 ms
   "2900RS001A01L01.FP_EN.AlarmDelay_H3" : Bool AT %DB5019.DBX47.7, 500 ms
   "2900RS001A01L01.FP_EN.AlarmDelay_H2" : Bool AT %DB5019.DBX48.0, 500 ms
   "2900RS001A01L01.FP_EN.AlarmDelay_H1" : Bool AT %DB5019.DBX48.1, 500 ms
   "2900RS001A01L01.FP_EN.AlarmDelay_L1" : Bool AT %DB5019.DBX48.2, 500 ms
   "2900RS001A01L01.FP_EN.AlarmDelay_L2" : Bool AT %DB5019.DBX48.3, 500 ms
   "2900RS001A01L01.FP_EN.AlarmDelay_L3" : Bool AT %DB5019.DBX48.4, 500 ms
   "2900RS001A01L01.FP_EN.ROC_Warn" : Bool AT %DB5019.DBX48.5, 500 ms
   "2900RS001A01L01.FP_EN.U_Range_Warn" : Bool AT %DB5019.DBX48.6, 500 ms
   "2900RS001A01L01.FP_EN.O_Range_Warn" : Bool AT %DB5019.DBX48.7, 500 ms
   "2900RS001A01L01.trend_tag_name" : TextRef, internal   // Еденицы измерения При експорте из ECS через скрипт - заполняется автоматически, если теги копируются в ручную то требуется задатать свойство Text - имя тега для тренда
   "2900RS001A01L01.DQ.AL_H3" : Bool AT %DB5019.DBX16.0, 500 ms
   "2900RS001A01L01.DQ.AL_H2" : Bool AT %DB5019.DBX16.1, 500 ms
   "2900RS001A01L01.DQ.AL_H1" : Bool AT %DB5019.DBX16.2, 500 ms
   "2900RS001A01L01.DQ.AL_L1" : Bool AT %DB5019.DBX16.3, 500 ms
   "2900RS001A01L01.DQ.AL_L2" : Bool AT %DB5019.DBX16.4, 500 ms
   "2900RS001A01L01.DQ.AL_L3" : Bool AT %DB5019.DBX16.5, 500 ms
   "2900RS001A01L01.DQ.SIG_OK" : Bool AT %DB5019.DBX16.6, 500 ms
   "2900RS001A01L01.DQ.LIM_H2" : Bool AT %DB5019.DBX16.7, 500 ms
   "2900RS001A01L01.DQ.LIM_H1" : Bool AT %DB5019.DBX17.0, 500 ms
   "2900RS001A01L01.DQ.LIM_L1" : Bool AT %DB5019.DBX17.1, 500 ms
   "2900RS001A01L01.DQ.LIM_L2" : Bool AT %DB5019.DBX17.2, 500 ms
   "2900RS001A01L01.DQ.GR_P" : Bool AT %DB5019.DBX17.3, 500 ms
   "2900RS001A01L01.DQ.GR_N" : Bool AT %DB5019.DBX17.4, 500 ms
   "2900RS001A01L01.I.IN" : Real AT %DB5019.DBD2, 500 ms
   "2900RS001A01L01.I.SIG_TYPE" : Int AT %DB5019.DBW0, 500 ms
   "2900RS001A01L01.I.FI_BUS" : Byte AT %DB5019.DBB6, 500 ms
   "2900RS001A01L01.DI.U_RANGE" : Bool AT %DB5019.DBX7.0, 500 ms
   "2900RS001A01L01.DI.O_RANGE" : Bool AT %DB5019.DBX7.1, 500 ms
   "2900RS001A01L01.DI.SIG_FAULT" : Bool AT %DB5019.DBX7.2, 500 ms
   "2900RS001A01L01.DI.EnConfig" : Bool AT %DB5019.DBX7.3, 500 ms
   "2900RS001A01L01.DI.AEN" : Bool AT %DB5019.DBX7.4, 500 ms
   "2900RS001A01L01.DI.AL_SUPR" : Bool AT %DB5019.DBX7.5, 500 ms
   "2900RS001A01L01.Q.PV_NORM" : Real AT %DB5019.DBD8, 500 ms
   "2900RS001A01L01.Q.PV_SCAL" : Real AT %DB5019.DBD12, 500 ms
   "2900RS001A01L01.ParentInfo" : TextRef, internal   // Имя родителя для попап окна, вкладка инфо. При експорте из ECS через скрипт заполняется автоматически, если теги копируются в ручную то требуется в ручную задатать свойство Start Value

HMI tags "2900RS001A01L02"
   "2900RS001A01L02.MSW" : 52809b66-421d-457f-8884-6f7a49d4e247 AT %DB5020.DBX18.0, 500 ms
   "2900RS001A01L02.DefaultText" : TextRef, internal   // Заголовок POPUP окна. При експорте из ECS через скрипт заполняется автоматически, если теги копируются в ручную то требуется в ручную задатать свойство Start Value
   "2900RS001A01L02.BlockInfo" : Array [0..2] of Int AT %DB5020.DBX38.0, 500 ms
   "2900RS001A01L02.StatusWork" : Int AT %DB5020.DBW242, 500 ms
   "2900RS001A01L02.FP_PARAM.DampingTime" : Int AT %DB5020.DBW50, 500 ms
   "2900RS001A01L02.FP_PARAM.Force_Value" : Real AT %DB5020.DBD52, 500 ms
   "2900RS001A01L02.FP_PARAM.Scale_Min" : Real AT %DB5020.DBD56, 500 ms
   "2900RS001A01L02.FP_PARAM.Scale_Max" : Real AT %DB5020.DBD60, 500 ms
   "2900RS001A01L02.FP_PARAM.Gradient" : Real AT %DB5020.DBD64, 500 ms
   "2900RS001A01L02.FP_PARAM.Grad_Pos" : Real AT %DB5020.DBD68, 500 ms
   "2900RS001A01L02.FP_PARAM.Grad_Neg" : Real AT %DB5020.DBD72, 500 ms
   "2900RS001A01L02.FP_PARAM.Grad_X" : Real AT %DB5020.DBD76, 500 ms
   "2900RS001A01L02.FP_PARAM.Gradient_Time_Pre" : Int AT %DB5020.DBW80, 500 ms
   "2900RS001A01L02.FP_PARAM.Gradient_Time_ACC" : Int AT %DB5020.DBW82, 500 ms
   "2900RS001A01L02.FP_PARAM.Alarm_Hyst" : Real AT %DB5020.DBD84, 500 ms
   "2900RS001A01L02.FP_PARAM.AlarmLimit_H3" : Real AT %DB5020.DBD88, 500 ms
   "2900RS001A01L02.FP_PARAM.AlarmLimit_H2" : Real AT %DB5020.DBD92, 500 ms
   "2900RS001A01L02.FP_PARAM.AlarmLimit_H1" : Real AT %DB5020.DBD96, 500 ms
   "2900RS001A01L02.FP_PARAM.AlarmLimit_L1" : Real AT %DB5020.DBD100, 500 ms
   "2900RS001A01L02.FP_PARAM.AlarmLimit_L2" : Real AT %DB5020.DBD104, 500 ms
   "2900RS001A01L02.FP_PARAM.AlarmLimit_L3" : Real AT %DB5020.DBD108, 500 ms
   "2900RS001A01L02.FP_PARAM.AlarmDelay_H3_Pre" : Int AT %DB5020.DBW112, 500 ms
   "2900RS001A01L02.FP_PARAM.AlarmDelay_H3_Acc" : Int AT %DB5020.DBW114, 500 ms
   "2900RS001A01L02.FP_PARAM.AlarmDelay_H2_Pre" : Int AT %DB5020.DBW116, 500 ms
   "2900RS001A01L02.FP_PARAM.AlarmDelay_H2_Acc" : Int AT %DB5020.DBW118, 500 ms
   "2900RS001A01L02.FP_PARAM.AlarmDelay_H1_Pre" : Int AT %DB5020.DBW120, 500 ms
   "2900RS001A01L02.FP_PARAM.AlarmDelay_H1_Acc" : Int AT %DB5020.DBW122, 500 ms
   "2900RS001A01L02.FP_PARAM.AlarmDelay_L1_Pre" : Int AT %DB5020.DBW124, 500 ms
   "2900RS001A01L02.FP_PARAM.AlarmDelay_L1_Acc" : Int AT %DB5020.DBW126, 500 ms
   "2900RS001A01L02.FP_PARAM.AlarmDelay_L2_Pre" : Int AT %DB5020.DBW128, 500 ms
   "2900RS001A01L02.FP_PARAM.AlarmDelay_L2_Acc" : Int AT %DB5020.DBW130, 500 ms
   "2900RS001A01L02.FP_PARAM.AlarmDelay_L3_Pre" : Int AT %DB5020.DBW132, 500 ms
   "2900RS001A01L02.FP_PARAM.AlarmDelay_L3_Acc" : Int AT %DB5020.DBW134, 500 ms
   "2900RS001A01L02.FP_PARAM.OpenLoopDelay_Pre" : Int AT %DB5020.DBW136, 500 ms
   "2900RS001A01L02.FP_PARAM.OpenLoopDelay_Acc" : Int AT %DB5020.DBW138, 500 ms
   "2900RS001A01L02.FP_PARAM.OverRangeDelay_Pre" : Int AT %DB5020.DBW140, 500 ms
   "2900RS001A01L02.FP_PARAM.OverRangeDelay_Acc" : Int AT %DB5020.DBW142, 500 ms
   "2900RS001A01L02.FP_PARAM.AuxLimit_H2_Value" : Real AT %DB5020.DBD144, 500 ms
   "2900RS001A01L02.FP_PARAM.AuxLimit_H1_Value" : Real AT %DB5020.DBD148, 500 ms
   "2900RS001A01L02.FP_PARAM.AuxLimit_L2_Value" : Real AT %DB5020.DBD152, 500 ms
   "2900RS001A01L02.FP_PARAM.AuxLimit_L1_Value" : Real AT %DB5020.DBD156, 500 ms
   "2900RS001A01L02.Unit" : TextRef, internal   // Еденицы измерения При експорте из ECS через скрипт заполняется автоматически, если теги копируются в ручную то требуется задатать свойство Text
   "2900RS001A01L02.Decimals" : TextRef, internal   // Формат отображения При експорте из ECS через скрипт, заполняется автоматически. Если теги копируются в ручную то требуется задатать свойство Text s999999.9
   "2900RS001A01L02.FP_EN.Square" : Bool AT %DB5020.DBX46.0, 500 ms
   "2900RS001A01L02.FP_EN.SquareRoot" : Bool AT %DB5020.DBX46.1, 500 ms
   "2900RS001A01L02.FP_EN.ParentSupress" : Bool AT %DB5020.DBX46.2, 500 ms
   "2900RS001A01L02.FP_EN.ParentSupressUnit" : Bool AT %DB5020.DBX46.3, 500 ms
   "2900RS001A01L02.FP_EN.Force" : Bool AT %DB5020.DBX46.4, 500 ms
   "2900RS001A01L02.FP_EN.Damping" : Bool AT %DB5020.DBX46.5, 500 ms
   "2900RS001A01L02.FP_EN.Gradient_Pos" : Bool AT %DB5020.DBX46.6, 500 ms
   "2900RS001A01L02.FP_EN.Gradient_Neg" : Bool AT %DB5020.DBX46.7, 500 ms
   "2900RS001A01L02.FP_EN.Hysteresis" : Bool AT %DB5020.DBX47.0, 500 ms
   "2900RS001A01L02.FP_EN.Alarm_H3" : Bool AT %DB5020.DBX47.1, 500 ms
   "2900RS001A01L02.FP_EN.Alarm_H2" : Bool AT %DB5020.DBX47.2, 500 ms
   "2900RS001A01L02.FP_EN.Alarm_H1" : Bool AT %DB5020.DBX47.3, 500 ms
   "2900RS001A01L02.FP_EN.Alarm_L1" : Bool AT %DB5020.DBX47.4, 500 ms
   "2900RS001A01L02.FP_EN.Alarm_L2" : Bool AT %DB5020.DBX47.5, 500 ms
   "2900RS001A01L02.FP_EN.Alarm_L3" : Bool AT %DB5020.DBX47.6, 500 ms
   "2900RS001A01L02.FP_EN.AlarmDelay_H3" : Bool AT %DB5020.DBX47.7, 500 ms
   "2900RS001A01L02.FP_EN.AlarmDelay_H2" : Bool AT %DB5020.DBX48.0, 500 ms
   "2900RS001A01L02.FP_EN.AlarmDelay_H1" : Bool AT %DB5020.DBX48.1, 500 ms
   "2900RS001A01L02.FP_EN.AlarmDelay_L1" : Bool AT %DB5020.DBX48.2, 500 ms
   "2900RS001A01L02.FP_EN.AlarmDelay_L2" : Bool AT %DB5020.DBX48.3, 500 ms
   "2900RS001A01L02.FP_EN.AlarmDelay_L3" : Bool AT %DB5020.DBX48.4, 500 ms
   "2900RS001A01L02.FP_EN.ROC_Warn" : Bool AT %DB5020.DBX48.5, 500 ms
   "2900RS001A01L02.FP_EN.U_Range_Warn" : Bool AT %DB5020.DBX48.6, 500 ms
   "2900RS001A01L02.FP_EN.O_Range_Warn" : Bool AT %DB5020.DBX48.7, 500 ms
   "2900RS001A01L02.trend_tag_name" : TextRef, internal   // Еденицы измерения При експорте из ECS через скрипт - заполняется автоматически, если теги копируются в ручную то требуется задатать свойство Text - имя тега для тренда
   "2900RS001A01L02.DQ.AL_H3" : Bool AT %DB5020.DBX16.0, 500 ms
   "2900RS001A01L02.DQ.AL_H2" : Bool AT %DB5020.DBX16.1, 500 ms
   "2900RS001A01L02.DQ.AL_H1" : Bool AT %DB5020.DBX16.2, 500 ms
   "2900RS001A01L02.DQ.AL_L1" : Bool AT %DB5020.DBX16.3, 500 ms
   "2900RS001A01L02.DQ.AL_L2" : Bool AT %DB5020.DBX16.4, 500 ms
   "2900RS001A01L02.DQ.AL_L3" : Bool AT %DB5020.DBX16.5, 500 ms
   "2900RS001A01L02.DQ.SIG_OK" : Bool AT %DB5020.DBX16.6, 500 ms
   "2900RS001A01L02.DQ.LIM_H2" : Bool AT %DB5020.DBX16.7, 500 ms
   "2900RS001A01L02.DQ.LIM_H1" : Bool AT %DB5020.DBX17.0, 500 ms
   "2900RS001A01L02.DQ.LIM_L1" : Bool AT %DB5020.DBX17.1, 500 ms
   "2900RS001A01L02.DQ.LIM_L2" : Bool AT %DB5020.DBX17.2, 500 ms
   "2900RS001A01L02.DQ.GR_P" : Bool AT %DB5020.DBX17.3, 500 ms
   "2900RS001A01L02.DQ.GR_N" : Bool AT %DB5020.DBX17.4, 500 ms
   "2900RS001A01L02.I.IN" : Real AT %DB5020.DBD2, 500 ms
   "2900RS001A01L02.I.SIG_TYPE" : Int AT %DB5020.DBW0, 500 ms
   "2900RS001A01L02.I.FI_BUS" : Byte AT %DB5020.DBB6, 500 ms
   "2900RS001A01L02.DI.U_RANGE" : Bool AT %DB5020.DBX7.0, 500 ms
   "2900RS001A01L02.DI.O_RANGE" : Bool AT %DB5020.DBX7.1, 500 ms
   "2900RS001A01L02.DI.SIG_FAULT" : Bool AT %DB5020.DBX7.2, 500 ms
   "2900RS001A01L02.DI.EnConfig" : Bool AT %DB5020.DBX7.3, 500 ms
   "2900RS001A01L02.DI.AEN" : Bool AT %DB5020.DBX7.4, 500 ms
   "2900RS001A01L02.DI.AL_SUPR" : Bool AT %DB5020.DBX7.5, 500 ms
   "2900RS001A01L02.Q.PV_NORM" : Real AT %DB5020.DBD8, 500 ms
   "2900RS001A01L02.Q.PV_SCAL" : Real AT %DB5020.DBD12, 500 ms
   "2900RS001A01L02.ParentInfo" : TextRef, internal   // Имя родителя для попап окна, вкладка инфо. При експорте из ECS через скрипт заполняется автоматически, если теги копируются в ручную то требуется в ручную задатать свойство Start Value

HMI tags "2900RS001A01L03"
   "2900RS001A01L03.MSW" : 52809b66-421d-457f-8884-6f7a49d4e247 AT %DB5021.DBX18.0, 500 ms
   "2900RS001A01L03.DefaultText" : TextRef, internal   // Заголовок POPUP окна. При експорте из ECS через скрипт заполняется автоматически, если теги копируются в ручную то требуется в ручную задатать свойство Start Value
   "2900RS001A01L03.BlockInfo" : Array [0..2] of Int AT %DB5021.DBX38.0, 500 ms
   "2900RS001A01L03.StatusWork" : Int AT %DB5021.DBW242, 500 ms
   "2900RS001A01L03.FP_PARAM.DampingTime" : Int AT %DB5021.DBW50, 500 ms
   "2900RS001A01L03.FP_PARAM.Force_Value" : Real AT %DB5021.DBD52, 500 ms
   "2900RS001A01L03.FP_PARAM.Scale_Min" : Real AT %DB5021.DBD56, 500 ms
   "2900RS001A01L03.FP_PARAM.Scale_Max" : Real AT %DB5021.DBD60, 500 ms
   "2900RS001A01L03.FP_PARAM.Gradient" : Real AT %DB5021.DBD64, 500 ms
   "2900RS001A01L03.FP_PARAM.Grad_Pos" : Real AT %DB5021.DBD68, 500 ms
   "2900RS001A01L03.FP_PARAM.Grad_Neg" : Real AT %DB5021.DBD72, 500 ms
   "2900RS001A01L03.FP_PARAM.Grad_X" : Real AT %DB5021.DBD76, 500 ms
   "2900RS001A01L03.FP_PARAM.Gradient_Time_Pre" : Int AT %DB5021.DBW80, 500 ms
   "2900RS001A01L03.FP_PARAM.Gradient_Time_ACC" : Int AT %DB5021.DBW82, 500 ms
   "2900RS001A01L03.FP_PARAM.Alarm_Hyst" : Real AT %DB5021.DBD84, 500 ms
   "2900RS001A01L03.FP_PARAM.AlarmLimit_H3" : Real AT %DB5021.DBD88, 500 ms
   "2900RS001A01L03.FP_PARAM.AlarmLimit_H2" : Real AT %DB5021.DBD92, 500 ms
   "2900RS001A01L03.FP_PARAM.AlarmLimit_H1" : Real AT %DB5021.DBD96, 500 ms
   "2900RS001A01L03.FP_PARAM.AlarmLimit_L1" : Real AT %DB5021.DBD100, 500 ms
   "2900RS001A01L03.FP_PARAM.AlarmLimit_L2" : Real AT %DB5021.DBD104, 500 ms
   "2900RS001A01L03.FP_PARAM.AlarmLimit_L3" : Real AT %DB5021.DBD108, 500 ms
   "2900RS001A01L03.FP_PARAM.AlarmDelay_H3_Pre" : Int AT %DB5021.DBW112, 500 ms
   "2900RS001A01L03.FP_PARAM.AlarmDelay_H3_Acc" : Int AT %DB5021.DBW114, 500 ms
   "2900RS001A01L03.FP_PARAM.AlarmDelay_H2_Pre" : Int AT %DB5021.DBW116, 500 ms
   "2900RS001A01L03.FP_PARAM.AlarmDelay_H2_Acc" : Int AT %DB5021.DBW118, 500 ms
   "2900RS001A01L03.FP_PARAM.AlarmDelay_H1_Pre" : Int AT %DB5021.DBW120, 500 ms
   "2900RS001A01L03.FP_PARAM.AlarmDelay_H1_Acc" : Int AT %DB5021.DBW122, 500 ms
   "2900RS001A01L03.FP_PARAM.AlarmDelay_L1_Pre" : Int AT %DB5021.DBW124, 500 ms
   "2900RS001A01L03.FP_PARAM.AlarmDelay_L1_Acc" : Int AT %DB5021.DBW126, 500 ms
   "2900RS001A01L03.FP_PARAM.AlarmDelay_L2_Pre" : Int AT %DB5021.DBW128, 500 ms
   "2900RS001A01L03.FP_PARAM.AlarmDelay_L2_Acc" : Int AT %DB5021.DBW130, 500 ms
   "2900RS001A01L03.FP_PARAM.AlarmDelay_L3_Pre" : Int AT %DB5021.DBW132, 500 ms
   "2900RS001A01L03.FP_PARAM.AlarmDelay_L3_Acc" : Int AT %DB5021.DBW134, 500 ms
   "2900RS001A01L03.FP_PARAM.OpenLoopDelay_Pre" : Int AT %DB5021.DBW136, 500 ms
   "2900RS001A01L03.FP_PARAM.OpenLoopDelay_Acc" : Int AT %DB5021.DBW138, 500 ms
   "2900RS001A01L03.FP_PARAM.OverRangeDelay_Pre" : Int AT %DB5021.DBW140, 500 ms
   "2900RS001A01L03.FP_PARAM.OverRangeDelay_Acc" : Int AT %DB5021.DBW142, 500 ms
   "2900RS001A01L03.FP_PARAM.AuxLimit_H2_Value" : Real AT %DB5021.DBD144, 500 ms
   "2900RS001A01L03.FP_PARAM.AuxLimit_H1_Value" : Real AT %DB5021.DBD148, 500 ms
   "2900RS001A01L03.FP_PARAM.AuxLimit_L2_Value" : Real AT %DB5021.DBD152, 500 ms
   "2900RS001A01L03.FP_PARAM.AuxLimit_L1_Value" : Real AT %DB5021.DBD156, 500 ms
   "2900RS001A01L03.Unit" : TextRef, internal   // Еденицы измерения При експорте из ECS через скрипт заполняется автоматически, если теги копируются в ручную то требуется задатать свойство Text
   "2900RS001A01L03.Decimals" : TextRef, internal   // Формат отображения При експорте из ECS через скрипт, заполняется автоматически. Если теги копируются в ручную то требуется задатать свойство Text s999999.9
   "2900RS001A01L03.FP_EN.Square" : Bool AT %DB5021.DBX46.0, 500 ms
   "2900RS001A01L03.FP_EN.SquareRoot" : Bool AT %DB5021.DBX46.1, 500 ms
   "2900RS001A01L03.FP_EN.ParentSupress" : Bool AT %DB5021.DBX46.2, 500 ms
   "2900RS001A01L03.FP_EN.ParentSupressUnit" : Bool AT %DB5021.DBX46.3, 500 ms
   "2900RS001A01L03.FP_EN.Force" : Bool AT %DB5021.DBX46.4, 500 ms
   "2900RS001A01L03.FP_EN.Damping" : Bool AT %DB5021.DBX46.5, 500 ms
   "2900RS001A01L03.FP_EN.Gradient_Pos" : Bool AT %DB5021.DBX46.6, 500 ms
   "2900RS001A01L03.FP_EN.Gradient_Neg" : Bool AT %DB5021.DBX46.7, 500 ms
   "2900RS001A01L03.FP_EN.Hysteresis" : Bool AT %DB5021.DBX47.0, 500 ms
   "2900RS001A01L03.FP_EN.Alarm_H3" : Bool AT %DB5021.DBX47.1, 500 ms
   "2900RS001A01L03.FP_EN.Alarm_H2" : Bool AT %DB5021.DBX47.2, 500 ms
   "2900RS001A01L03.FP_EN.Alarm_H1" : Bool AT %DB5021.DBX47.3, 500 ms
   "2900RS001A01L03.FP_EN.Alarm_L1" : Bool AT %DB5021.DBX47.4, 500 ms
   "2900RS001A01L03.FP_EN.Alarm_L2" : Bool AT %DB5021.DBX47.5, 500 ms
   "2900RS001A01L03.FP_EN.Alarm_L3" : Bool AT %DB5021.DBX47.6, 500 ms
   "2900RS001A01L03.FP_EN.AlarmDelay_H3" : Bool AT %DB5021.DBX47.7, 500 ms
   "2900RS001A01L03.FP_EN.AlarmDelay_H2" : Bool AT %DB5021.DBX48.0, 500 ms
   "2900RS001A01L03.FP_EN.AlarmDelay_H1" : Bool AT %DB5021.DBX48.1, 500 ms
   "2900RS001A01L03.FP_EN.AlarmDelay_L1" : Bool AT %DB5021.DBX48.2, 500 ms
   "2900RS001A01L03.FP_EN.AlarmDelay_L2" : Bool AT %DB5021.DBX48.3, 500 ms
   "2900RS001A01L03.FP_EN.AlarmDelay_L3" : Bool AT %DB5021.DBX48.4, 500 ms
   "2900RS001A01L03.FP_EN.ROC_Warn" : Bool AT %DB5021.DBX48.5, 500 ms
   "2900RS001A01L03.FP_EN.U_Range_Warn" : Bool AT %DB5021.DBX48.6, 500 ms
   "2900RS001A01L03.FP_EN.O_Range_Warn" : Bool AT %DB5021.DBX48.7, 500 ms
   "2900RS001A01L03.trend_tag_name" : TextRef, internal   // Еденицы измерения При експорте из ECS через скрипт - заполняется автоматически, если теги копируются в ручную то требуется задатать свойство Text - имя тега для тренда
   "2900RS001A01L03.DQ.AL_H3" : Bool AT %DB5021.DBX16.0, 500 ms
   "2900RS001A01L03.DQ.AL_H2" : Bool AT %DB5021.DBX16.1, 500 ms
   "2900RS001A01L03.DQ.AL_H1" : Bool AT %DB5021.DBX16.2, 500 ms
   "2900RS001A01L03.DQ.AL_L1" : Bool AT %DB5021.DBX16.3, 500 ms
   "2900RS001A01L03.DQ.AL_L2" : Bool AT %DB5021.DBX16.4, 500 ms
   "2900RS001A01L03.DQ.AL_L3" : Bool AT %DB5021.DBX16.5, 500 ms
   "2900RS001A01L03.DQ.SIG_OK" : Bool AT %DB5021.DBX16.6, 500 ms
   "2900RS001A01L03.DQ.LIM_H2" : Bool AT %DB5021.DBX16.7, 500 ms
   "2900RS001A01L03.DQ.LIM_H1" : Bool AT %DB5021.DBX17.0, 500 ms
   "2900RS001A01L03.DQ.LIM_L1" : Bool AT %DB5021.DBX17.1, 500 ms
   "2900RS001A01L03.DQ.LIM_L2" : Bool AT %DB5021.DBX17.2, 500 ms
   "2900RS001A01L03.DQ.GR_P" : Bool AT %DB5021.DBX17.3, 500 ms
   "2900RS001A01L03.DQ.GR_N" : Bool AT %DB5021.DBX17.4, 500 ms
   "2900RS001A01L03.I.IN" : Real AT %DB5021.DBD2, 500 ms
   "2900RS001A01L03.I.SIG_TYPE" : Int AT %DB5021.DBW0, 500 ms
   "2900RS001A01L03.I.FI_BUS" : Byte AT %DB5021.DBB6, 500 ms
   "2900RS001A01L03.DI.U_RANGE" : Bool AT %DB5021.DBX7.0, 500 ms
   "2900RS001A01L03.DI.O_RANGE" : Bool AT %DB5021.DBX7.1, 500 ms
   "2900RS001A01L03.DI.SIG_FAULT" : Bool AT %DB5021.DBX7.2, 500 ms
   "2900RS001A01L03.DI.EnConfig" : Bool AT %DB5021.DBX7.3, 500 ms
   "2900RS001A01L03.DI.AEN" : Bool AT %DB5021.DBX7.4, 500 ms
   "2900RS001A01L03.DI.AL_SUPR" : Bool AT %DB5021.DBX7.5, 500 ms
   "2900RS001A01L03.Q.PV_NORM" : Real AT %DB5021.DBD8, 500 ms
   "2900RS001A01L03.Q.PV_SCAL" : Real AT %DB5021.DBD12, 500 ms
   "2900RS001A01L03.ParentInfo" : TextRef, internal   // Имя родителя для попап окна, вкладка инфо. При експорте из ECS через скрипт заполняется автоматически, если теги копируются в ручную то требуется в ручную задатать свойство Start Value

HMI tags "2900RS001A01T02"
   "2900RS001A01T02.MSW" : 52809b66-421d-457f-8884-6f7a49d4e247 AT %DB5022.DBX18.0, 500 ms
   "2900RS001A01T02.DefaultText" : TextRef, internal   // Заголовок POPUP окна. При експорте из ECS через скрипт заполняется автоматически, если теги копируются в ручную то требуется в ручную задатать свойство Start Value
   "2900RS001A01T02.BlockInfo" : Array [0..2] of Int AT %DB5022.DBX38.0, 500 ms
   "2900RS001A01T02.StatusWork" : Int AT %DB5022.DBW242, 500 ms
   "2900RS001A01T02.FP_PARAM.DampingTime" : Int AT %DB5022.DBW50, 500 ms
   "2900RS001A01T02.FP_PARAM.Force_Value" : Real AT %DB5022.DBD52, 500 ms
   "2900RS001A01T02.FP_PARAM.Scale_Min" : Real AT %DB5022.DBD56, 500 ms
   "2900RS001A01T02.FP_PARAM.Scale_Max" : Real AT %DB5022.DBD60, 500 ms
   "2900RS001A01T02.FP_PARAM.Gradient" : Real AT %DB5022.DBD64, 500 ms
   "2900RS001A01T02.FP_PARAM.Grad_Pos" : Real AT %DB5022.DBD68, 500 ms
   "2900RS001A01T02.FP_PARAM.Grad_Neg" : Real AT %DB5022.DBD72, 500 ms
   "2900RS001A01T02.FP_PARAM.Grad_X" : Real AT %DB5022.DBD76, 500 ms
   "2900RS001A01T02.FP_PARAM.Gradient_Time_Pre" : Int AT %DB5022.DBW80, 500 ms
   "2900RS001A01T02.FP_PARAM.Gradient_Time_ACC" : Int AT %DB5022.DBW82, 500 ms
   "2900RS001A01T02.FP_PARAM.Alarm_Hyst" : Real AT %DB5022.DBD84, 500 ms
   "2900RS001A01T02.FP_PARAM.AlarmLimit_H3" : Real AT %DB5022.DBD88, 500 ms
   "2900RS001A01T02.FP_PARAM.AlarmLimit_H2" : Real AT %DB5022.DBD92, 500 ms
   "2900RS001A01T02.FP_PARAM.AlarmLimit_H1" : Real AT %DB5022.DBD96, 500 ms
   "2900RS001A01T02.FP_PARAM.AlarmLimit_L1" : Real AT %DB5022.DBD100, 500 ms
   "2900RS001A01T02.FP_PARAM.AlarmLimit_L2" : Real AT %DB5022.DBD104, 500 ms
   "2900RS001A01T02.FP_PARAM.AlarmLimit_L3" : Real AT %DB5022.DBD108, 500 ms
   "2900RS001A01T02.FP_PARAM.AlarmDelay_H3_Pre" : Int AT %DB5022.DBW112, 500 ms
   "2900RS001A01T02.FP_PARAM.AlarmDelay_H3_Acc" : Int AT %DB5022.DBW114, 500 ms
   "2900RS001A01T02.FP_PARAM.AlarmDelay_H2_Pre" : Int AT %DB5022.DBW116, 500 ms
   "2900RS001A01T02.FP_PARAM.AlarmDelay_H2_Acc" : Int AT %DB5022.DBW118, 500 ms
   "2900RS001A01T02.FP_PARAM.AlarmDelay_H1_Pre" : Int AT %DB5022.DBW120, 500 ms
   "2900RS001A01T02.FP_PARAM.AlarmDelay_H1_Acc" : Int AT %DB5022.DBW122, 500 ms
   "2900RS001A01T02.FP_PARAM.AlarmDelay_L1_Pre" : Int AT %DB5022.DBW124, 500 ms
   "2900RS001A01T02.FP_PARAM.AlarmDelay_L1_Acc" : Int AT %DB5022.DBW126, 500 ms
   "2900RS001A01T02.FP_PARAM.AlarmDelay_L2_Pre" : Int AT %DB5022.DBW128, 500 ms
   "2900RS001A01T02.FP_PARAM.AlarmDelay_L2_Acc" : Int AT %DB5022.DBW130, 500 ms
   "2900RS001A01T02.FP_PARAM.AlarmDelay_L3_Pre" : Int AT %DB5022.DBW132, 500 ms
   "2900RS001A01T02.FP_PARAM.AlarmDelay_L3_Acc" : Int AT %DB5022.DBW134, 500 ms
   "2900RS001A01T02.FP_PARAM.OpenLoopDelay_Pre" : Int AT %DB5022.DBW136, 500 ms
   "2900RS001A01T02.FP_PARAM.OpenLoopDelay_Acc" : Int AT %DB5022.DBW138, 500 ms
   "2900RS001A01T02.FP_PARAM.OverRangeDelay_Pre" : Int AT %DB5022.DBW140, 500 ms
   "2900RS001A01T02.FP_PARAM.OverRangeDelay_Acc" : Int AT %DB5022.DBW142, 500 ms
   "2900RS001A01T02.FP_PARAM.AuxLimit_H2_Value" : Real AT %DB5022.DBD144, 500 ms
   "2900RS001A01T02.FP_PARAM.AuxLimit_H1_Value" : Real AT %DB5022.DBD148, 500 ms
   "2900RS001A01T02.FP_PARAM.AuxLimit_L2_Value" : Real AT %DB5022.DBD152, 500 ms
   "2900RS001A01T02.FP_PARAM.AuxLimit_L1_Value" : Real AT %DB5022.DBD156, 500 ms
   "2900RS001A01T02.Unit" : TextRef, internal   // Еденицы измерения При експорте из ECS через скрипт заполняется автоматически, если теги копируются в ручную то требуется задатать свойство Text
   "2900RS001A01T02.Decimals" : TextRef, internal   // Формат отображения При експорте из ECS через скрипт, заполняется автоматически. Если теги копируются в ручную то требуется задатать свойство Text s999999.9
   "2900RS001A01T02.FP_EN.Square" : Bool AT %DB5022.DBX46.0, 500 ms
   "2900RS001A01T02.FP_EN.SquareRoot" : Bool AT %DB5022.DBX46.1, 500 ms
   "2900RS001A01T02.FP_EN.ParentSupress" : Bool AT %DB5022.DBX46.2, 500 ms
   "2900RS001A01T02.FP_EN.ParentSupressUnit" : Bool AT %DB5022.DBX46.3, 500 ms
   "2900RS001A01T02.FP_EN.Force" : Bool AT %DB5022.DBX46.4, 500 ms
   "2900RS001A01T02.FP_EN.Damping" : Bool AT %DB5022.DBX46.5, 500 ms
   "2900RS001A01T02.FP_EN.Gradient_Pos" : Bool AT %DB5022.DBX46.6, 500 ms
   "2900RS001A01T02.FP_EN.Gradient_Neg" : Bool AT %DB5022.DBX46.7, 500 ms
   "2900RS001A01T02.FP_EN.Hysteresis" : Bool AT %DB5022.DBX47.0, 500 ms
   "2900RS001A01T02.FP_EN.Alarm_H3" : Bool AT %DB5022.DBX47.1, 500 ms
   "2900RS001A01T02.FP_EN.Alarm_H2" : Bool AT %DB5022.DBX47.2, 500 ms
   "2900RS001A01T02.FP_EN.Alarm_H1" : Bool AT %DB5022.DBX47.3, 500 ms
   "2900RS001A01T02.FP_EN.Alarm_L1" : Bool AT %DB5022.DBX47.4, 500 ms
   "2900RS001A01T02.FP_EN.Alarm_L2" : Bool AT %DB5022.DBX47.5, 500 ms
   "2900RS001A01T02.FP_EN.Alarm_L3" : Bool AT %DB5022.DBX47.6, 500 ms
   "2900RS001A01T02.FP_EN.AlarmDelay_H3" : Bool AT %DB5022.DBX47.7, 500 ms
   "2900RS001A01T02.FP_EN.AlarmDelay_H2" : Bool AT %DB5022.DBX48.0, 500 ms
   "2900RS001A01T02.FP_EN.AlarmDelay_H1" : Bool AT %DB5022.DBX48.1, 500 ms
   "2900RS001A01T02.FP_EN.AlarmDelay_L1" : Bool AT %DB5022.DBX48.2, 500 ms
   "2900RS001A01T02.FP_EN.AlarmDelay_L2" : Bool AT %DB5022.DBX48.3, 500 ms
   "2900RS001A01T02.FP_EN.AlarmDelay_L3" : Bool AT %DB5022.DBX48.4, 500 ms
   "2900RS001A01T02.FP_EN.ROC_Warn" : Bool AT %DB5022.DBX48.5, 500 ms
   "2900RS001A01T02.FP_EN.U_Range_Warn" : Bool AT %DB5022.DBX48.6, 500 ms
   "2900RS001A01T02.FP_EN.O_Range_Warn" : Bool AT %DB5022.DBX48.7, 500 ms
   "2900RS001A01T02.trend_tag_name" : TextRef, internal   // Еденицы измерения При експорте из ECS через скрипт - заполняется автоматически, если теги копируются в ручную то требуется задатать свойство Text - имя тега для тренда
   "2900RS001A01T02.DQ.AL_H3" : Bool AT %DB5022.DBX16.0, 500 ms
   "2900RS001A01T02.DQ.AL_H2" : Bool AT %DB5022.DBX16.1, 500 ms
   "2900RS001A01T02.DQ.AL_H1" : Bool AT %DB5022.DBX16.2, 500 ms
   "2900RS001A01T02.DQ.AL_L1" : Bool AT %DB5022.DBX16.3, 500 ms
   "2900RS001A01T02.DQ.AL_L2" : Bool AT %DB5022.DBX16.4, 500 ms
   "2900RS001A01T02.DQ.AL_L3" : Bool AT %DB5022.DBX16.5, 500 ms
   "2900RS001A01T02.DQ.SIG_OK" : Bool AT %DB5022.DBX16.6, 500 ms
   "2900RS001A01T02.DQ.LIM_H2" : Bool AT %DB5022.DBX16.7, 500 ms
   "2900RS001A01T02.DQ.LIM_H1" : Bool AT %DB5022.DBX17.0, 500 ms
   "2900RS001A01T02.DQ.LIM_L1" : Bool AT %DB5022.DBX17.1, 500 ms
   "2900RS001A01T02.DQ.LIM_L2" : Bool AT %DB5022.DBX17.2, 500 ms
   "2900RS001A01T02.DQ.GR_P" : Bool AT %DB5022.DBX17.3, 500 ms
   "2900RS001A01T02.DQ.GR_N" : Bool AT %DB5022.DBX17.4, 500 ms
   "2900RS001A01T02.I.IN" : Real AT %DB5022.DBD2, 500 ms
   "2900RS001A01T02.I.SIG_TYPE" : Int AT %DB5022.DBW0, 500 ms
   "2900RS001A01T02.I.FI_BUS" : Byte AT %DB5022.DBB6, 500 ms
   "2900RS001A01T02.DI.U_RANGE" : Bool AT %DB5022.DBX7.0, 500 ms
   "2900RS001A01T02.DI.O_RANGE" : Bool AT %DB5022.DBX7.1, 500 ms
   "2900RS001A01T02.DI.SIG_FAULT" : Bool AT %DB5022.DBX7.2, 500 ms
   "2900RS001A01T02.DI.EnConfig" : Bool AT %DB5022.DBX7.3, 500 ms
   "2900RS001A01T02.DI.AEN" : Bool AT %DB5022.DBX7.4, 500 ms
   "2900RS001A01T02.DI.AL_SUPR" : Bool AT %DB5022.DBX7.5, 500 ms
   "2900RS001A01T02.Q.PV_NORM" : Real AT %DB5022.DBD8, 500 ms
   "2900RS001A01T02.Q.PV_SCAL" : Real AT %DB5022.DBD12, 500 ms
   "2900RS001A01T02.ParentInfo" : TextRef, internal   // Имя родителя для попап окна, вкладка инфо. При експорте из ECS через скрипт заполняется автоматически, если теги копируются в ручную то требуется в ручную задатать свойство Start Value

HMI tags "2905RS001A01F01"
   "2905RS001A01F01.MSW" : 52809b66-421d-457f-8884-6f7a49d4e247 AT %DB5023.DBX18.0, 500 ms
   "2905RS001A01F01.DefaultText" : TextRef, internal   // Заголовок POPUP окна. При експорте из ECS через скрипт заполняется автоматически, если теги копируются в ручную то требуется в ручную задатать свойство Start Value
   "2905RS001A01F01.BlockInfo" : Array [0..2] of Int AT %DB5023.DBX38.0, 500 ms
   "2905RS001A01F01.StatusWork" : Int AT %DB5023.DBW242, 500 ms
   "2905RS001A01F01.FP_PARAM.DampingTime" : Int AT %DB5023.DBW50, 500 ms
   "2905RS001A01F01.FP_PARAM.Force_Value" : Real AT %DB5023.DBD52, 500 ms
   "2905RS001A01F01.FP_PARAM.Scale_Min" : Real AT %DB5023.DBD56, 500 ms
   "2905RS001A01F01.FP_PARAM.Scale_Max" : Real AT %DB5023.DBD60, 500 ms
   "2905RS001A01F01.FP_PARAM.Gradient" : Real AT %DB5023.DBD64, 500 ms
   "2905RS001A01F01.FP_PARAM.Grad_Pos" : Real AT %DB5023.DBD68, 500 ms
   "2905RS001A01F01.FP_PARAM.Grad_Neg" : Real AT %DB5023.DBD72, 500 ms
   "2905RS001A01F01.FP_PARAM.Grad_X" : Real AT %DB5023.DBD76, 500 ms
   "2905RS001A01F01.FP_PARAM.Gradient_Time_Pre" : Int AT %DB5023.DBW80, 500 ms
   "2905RS001A01F01.FP_PARAM.Gradient_Time_ACC" : Int AT %DB5023.DBW82, 500 ms
   "2905RS001A01F01.FP_PARAM.Alarm_Hyst" : Real AT %DB5023.DBD84, 500 ms
   "2905RS001A01F01.FP_PARAM.AlarmLimit_H3" : Real AT %DB5023.DBD88, 500 ms
   "2905RS001A01F01.FP_PARAM.AlarmLimit_H2" : Real AT %DB5023.DBD92, 500 ms
   "2905RS001A01F01.FP_PARAM.AlarmLimit_H1" : Real AT %DB5023.DBD96, 500 ms
   "2905RS001A01F01.FP_PARAM.AlarmLimit_L1" : Real AT %DB5023.DBD100, 500 ms
   "2905RS001A01F01.FP_PARAM.AlarmLimit_L2" : Real AT %DB5023.DBD104, 500 ms
   "2905RS001A01F01.FP_PARAM.AlarmLimit_L3" : Real AT %DB5023.DBD108, 500 ms
   "2905RS001A01F01.FP_PARAM.AlarmDelay_H3_Pre" : Int AT %DB5023.DBW112, 500 ms
   "2905RS001A01F01.FP_PARAM.AlarmDelay_H3_Acc" : Int AT %DB5023.DBW114, 500 ms
   "2905RS001A01F01.FP_PARAM.AlarmDelay_H2_Pre" : Int AT %DB5023.DBW116, 500 ms
   "2905RS001A01F01.FP_PARAM.AlarmDelay_H2_Acc" : Int AT %DB5023.DBW118, 500 ms
   "2905RS001A01F01.FP_PARAM.AlarmDelay_H1_Pre" : Int AT %DB5023.DBW120, 500 ms
   "2905RS001A01F01.FP_PARAM.AlarmDelay_H1_Acc" : Int AT %DB5023.DBW122, 500 ms
   "2905RS001A01F01.FP_PARAM.AlarmDelay_L1_Pre" : Int AT %DB5023.DBW124, 500 ms
   "2905RS001A01F01.FP_PARAM.AlarmDelay_L1_Acc" : Int AT %DB5023.DBW126, 500 ms
   "2905RS001A01F01.FP_PARAM.AlarmDelay_L2_Pre" : Int AT %DB5023.DBW128, 500 ms
   "2905RS001A01F01.FP_PARAM.AlarmDelay_L2_Acc" : Int AT %DB5023.DBW130, 500 ms
   "2905RS001A01F01.FP_PARAM.AlarmDelay_L3_Pre" : Int AT %DB5023.DBW132, 500 ms
   "2905RS001A01F01.FP_PARAM.AlarmDelay_L3_Acc" : Int AT %DB5023.DBW134, 500 ms
   "2905RS001A01F01.FP_PARAM.OpenLoopDelay_Pre" : Int AT %DB5023.DBW136, 500 ms
   "2905RS001A01F01.FP_PARAM.OpenLoopDelay_Acc" : Int AT %DB5023.DBW138, 500 ms
   "2905RS001A01F01.FP_PARAM.OverRangeDelay_Pre" : Int AT %DB5023.DBW140, 500 ms
   "2905RS001A01F01.FP_PARAM.OverRangeDelay_Acc" : Int AT %DB5023.DBW142, 500 ms
   "2905RS001A01F01.FP_PARAM.AuxLimit_H2_Value" : Real AT %DB5023.DBD144, 500 ms
   "2905RS001A01F01.FP_PARAM.AuxLimit_H1_Value" : Real AT %DB5023.DBD148, 500 ms
   "2905RS001A01F01.FP_PARAM.AuxLimit_L2_Value" : Real AT %DB5023.DBD152, 500 ms
   "2905RS001A01F01.FP_PARAM.AuxLimit_L1_Value" : Real AT %DB5023.DBD156, 500 ms
   "2905RS001A01F01.Unit" : TextRef, internal   // Еденицы измерения При експорте из ECS через скрипт заполняется автоматически, если теги копируются в ручную то требуется задатать свойство Text
   "2905RS001A01F01.Decimals" : TextRef, internal   // Формат отображения При експорте из ECS через скрипт, заполняется автоматически. Если теги копируются в ручную то требуется задатать свойство Text s999999.9
   "2905RS001A01F01.FP_EN.Square" : Bool AT %DB5023.DBX46.0, 500 ms
   "2905RS001A01F01.FP_EN.SquareRoot" : Bool AT %DB5023.DBX46.1, 500 ms
   "2905RS001A01F01.FP_EN.ParentSupress" : Bool AT %DB5023.DBX46.2, 500 ms
   "2905RS001A01F01.FP_EN.ParentSupressUnit" : Bool AT %DB5023.DBX46.3, 500 ms
   "2905RS001A01F01.FP_EN.Force" : Bool AT %DB5023.DBX46.4, 500 ms
   "2905RS001A01F01.FP_EN.Damping" : Bool AT %DB5023.DBX46.5, 500 ms
   "2905RS001A01F01.FP_EN.Gradient_Pos" : Bool AT %DB5023.DBX46.6, 500 ms
   "2905RS001A01F01.FP_EN.Gradient_Neg" : Bool AT %DB5023.DBX46.7, 500 ms
   "2905RS001A01F01.FP_EN.Hysteresis" : Bool AT %DB5023.DBX47.0, 500 ms
   "2905RS001A01F01.FP_EN.Alarm_H3" : Bool AT %DB5023.DBX47.1, 500 ms
   "2905RS001A01F01.FP_EN.Alarm_H2" : Bool AT %DB5023.DBX47.2, 500 ms
   "2905RS001A01F01.FP_EN.Alarm_H1" : Bool AT %DB5023.DBX47.3, 500 ms
   "2905RS001A01F01.FP_EN.Alarm_L1" : Bool AT %DB5023.DBX47.4, 500 ms
   "2905RS001A01F01.FP_EN.Alarm_L2" : Bool AT %DB5023.DBX47.5, 500 ms
   "2905RS001A01F01.FP_EN.Alarm_L3" : Bool AT %DB5023.DBX47.6, 500 ms
   "2905RS001A01F01.FP_EN.AlarmDelay_H3" : Bool AT %DB5023.DBX47.7, 500 ms
   "2905RS001A01F01.FP_EN.AlarmDelay_H2" : Bool AT %DB5023.DBX48.0, 500 ms
   "2905RS001A01F01.FP_EN.AlarmDelay_H1" : Bool AT %DB5023.DBX48.1, 500 ms
   "2905RS001A01F01.FP_EN.AlarmDelay_L1" : Bool AT %DB5023.DBX48.2, 500 ms
   "2905RS001A01F01.FP_EN.AlarmDelay_L2" : Bool AT %DB5023.DBX48.3, 500 ms
   "2905RS001A01F01.FP_EN.AlarmDelay_L3" : Bool AT %DB5023.DBX48.4, 500 ms
   "2905RS001A01F01.FP_EN.ROC_Warn" : Bool AT %DB5023.DBX48.5, 500 ms
   "2905RS001A01F01.FP_EN.U_Range_Warn" : Bool AT %DB5023.DBX48.6, 500 ms
   "2905RS001A01F01.FP_EN.O_Range_Warn" : Bool AT %DB5023.DBX48.7, 500 ms
   "2905RS001A01F01.trend_tag_name" : TextRef, internal   // Еденицы измерения При експорте из ECS через скрипт - заполняется автоматически, если теги копируются в ручную то требуется задатать свойство Text - имя тега для тренда
   "2905RS001A01F01.DQ.AL_H3" : Bool AT %DB5023.DBX16.0, 500 ms
   "2905RS001A01F01.DQ.AL_H2" : Bool AT %DB5023.DBX16.1, 500 ms
   "2905RS001A01F01.DQ.AL_H1" : Bool AT %DB5023.DBX16.2, 500 ms
   "2905RS001A01F01.DQ.AL_L1" : Bool AT %DB5023.DBX16.3, 500 ms
   "2905RS001A01F01.DQ.AL_L2" : Bool AT %DB5023.DBX16.4, 500 ms
   "2905RS001A01F01.DQ.AL_L3" : Bool AT %DB5023.DBX16.5, 500 ms
   "2905RS001A01F01.DQ.SIG_OK" : Bool AT %DB5023.DBX16.6, 500 ms
   "2905RS001A01F01.DQ.LIM_H2" : Bool AT %DB5023.DBX16.7, 500 ms
   "2905RS001A01F01.DQ.LIM_H1" : Bool AT %DB5023.DBX17.0, 500 ms
   "2905RS001A01F01.DQ.LIM_L1" : Bool AT %DB5023.DBX17.1, 500 ms
   "2905RS001A01F01.DQ.LIM_L2" : Bool AT %DB5023.DBX17.2, 500 ms
   "2905RS001A01F01.DQ.GR_P" : Bool AT %DB5023.DBX17.3, 500 ms
   "2905RS001A01F01.DQ.GR_N" : Bool AT %DB5023.DBX17.4, 500 ms
   "2905RS001A01F01.I.IN" : Real AT %DB5023.DBD2, 500 ms
   "2905RS001A01F01.I.SIG_TYPE" : Int AT %DB5023.DBW0, 500 ms
   "2905RS001A01F01.I.FI_BUS" : Byte AT %DB5023.DBB6, 500 ms
   "2905RS001A01F01.DI.U_RANGE" : Bool AT %DB5023.DBX7.0, 500 ms
   "2905RS001A01F01.DI.O_RANGE" : Bool AT %DB5023.DBX7.1, 500 ms
   "2905RS001A01F01.DI.SIG_FAULT" : Bool AT %DB5023.DBX7.2, 500 ms
   "2905RS001A01F01.DI.EnConfig" : Bool AT %DB5023.DBX7.3, 500 ms
   "2905RS001A01F01.DI.AEN" : Bool AT %DB5023.DBX7.4, 500 ms
   "2905RS001A01F01.DI.AL_SUPR" : Bool AT %DB5023.DBX7.5, 500 ms
   "2905RS001A01F01.Q.PV_NORM" : Real AT %DB5023.DBD8, 500 ms
   "2905RS001A01F01.Q.PV_SCAL" : Real AT %DB5023.DBD12, 500 ms
   "2905RS001A01F01.ParentInfo" : TextRef, internal   // Имя родителя для попап окна, вкладка инфо. При експорте из ECS через скрипт заполняется автоматически, если теги копируются в ручную то требуется в ручную задатать свойство Start Value

